KUKA KRL program: MyProgram_306().src

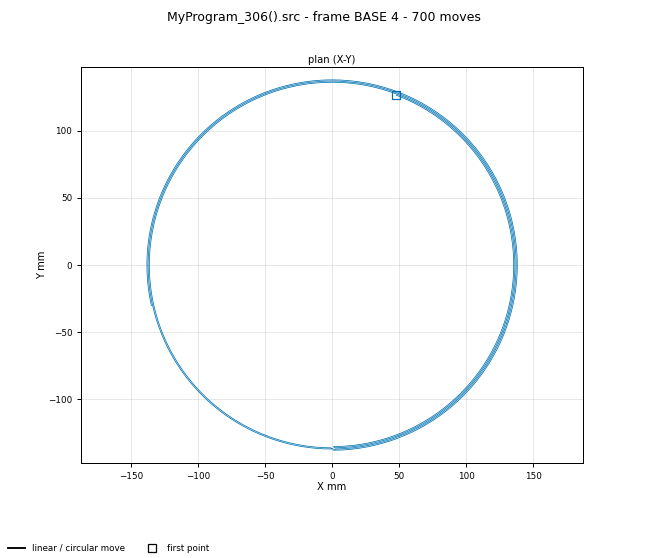
[picture p0: tool path of MyProgram_306().src in frame BASE 4, 700 of 700 moves have a stored position in this frame; points joined in program order, loops and branches not executed]
&ACCESS RVP
&REL 1
&PARAM TEMPLATE = C:\KRC\Roboter\Template\vorgabe
&PARAM EDITMASK = *
DEF MyProgram_306()
; ---- Setting reference (Base) ----
$BASE = BASE_DATA[4]

; --------------------------
; ---- Setting tool (TCP) ----
$TOOL = TOOL_DATA[3]
; --------------------------

$VEL.CP = VEL_APROX_PRINT
Startdeposition()
$VEL.CP = VEL_PRINT
LIN {X 47.8196,Y 126.5407,Z 181,A 70.0774,B 5.1523,C 0.0981,E1 5.2125,E2 382.635} C_DIS
LIN {X 50.7424,Y 125.3967,Z 181,A 68.7404,B 5.1523,C 0.0996,E1 5.216,E2 383.9727} C_DIS
LIN {X 53.7294,Y 124.1461,Z 181,A 67.3289,B 5.1523,C 0.1017,E1 5.2196,E2 385.3889} C_DIS
LIN {X 56.8494,Y 122.7487,Z 181,A 65.9585,B 5.1523,C 0.1025,E1 5.2231,E2 386.7498} C_DIS
LIN {X 60.1099,Y 121.1856,Z 181,A 64.4144,B 5.1522,C 0.1046,E1 5.227,E2 388.2953} C_DIS
LIN {X 63.2317,Y 119.5867,Z 181,A 62.9237,B 5.1522,C 0.1067,E1 5.2307,E2 389.7866} C_DIS
LIN {X 66.7997,Y 117.6329,Z 181,A 61.188,B 5.1522,C 0.1093,E1 5.2349,E2 391.5239} C_DIS
LIN {X 70.4878,Y 115.4608,Z 181,A 59.3984,B 5.152,C 0.1117,E1 5.2392,E2 393.3106} C_DIS
LIN {X 74.0978,Y 113.178,Z 181,A 57.6415,B 5.152,C 0.1139,E1 5.2433,E2 395.0613} C_DIS
LIN {X 77.4734,Y 110.8944,Z 181,A 55.903,B 5.152,C 0.1169,E1 5.2473,E2 396.8013} C_DIS
LIN {X 81.0975,Y 108.2727,Z 181,A 54.0011,B 5.1519,C 0.1202,E1 5.2516,E2 398.7043} C_DIS
LIN {X 84.4536,Y 105.6754,Z 181,A 52.2027,B 5.1518,C 0.1234,E1 5.2555,E2 400.5031} C_DIS
LIN {X 88.093,Y 102.6611,Z 181,A 50.2728,B 5.1518,C 0.1262,E1 5.2597,E2 402.4245} C_DIS
LIN {X 93.5773,Y 97.6879,Z 181,A 47.5115,B 5.1517,C 0.1274,E1 5.2653,E2 405.1411} C_DIS
LIN {X 95.6512,Y 95.6591,Z 181,A 45.6814,B 5.1514,C 0.1378,E1 5.269,E2 407.0442} C_DIS
LIN {X 98.4319,Y 92.7943,Z 181,A 44.4153,B 5.1514,C 0.1357,E1 5.2714,E2 408.2594} C_DIS
LIN {X 101.2138,Y 89.752,Z 181,A 42.6533,B 5.1514,C 0.1396,E1 5.2746,E2 410.0238} C_DIS
LIN {X 104.2851,Y 86.1641,Z 181,A 40.6959,B 5.1513,C 0.1434,E1 5.2782,E2 411.9765} C_DIS
LIN {X 107.3098,Y 82.3668,Z 181,A 38.7925,B 5.1512,C 0.146,E1 5.2814,E2 413.8619} C_DIS
LIN {X 109.5448,Y 79.3698,Z 181,A 37.1257,B 5.1511,C 0.1508,E1 5.2842,E2 415.5394} C_DIS
LIN {X 112.0158,Y 75.8426,Z 181,A 35.3544,B 5.151,C 0.1543,E1 5.287,E2 417.3049} C_DIS
LIN {X 114.5681,Y 71.9297,Z 181,A 33.411,B 5.1508,C 0.1586,E1 5.2899,E2 419.2447} C_DIS
LIN {X 116.9119,Y 68.0539,Z 181,A 31.5375,B 5.1507,C 0.1627,E1 5.2926,E2 421.1136} C_DIS
LIN {X 119.0066,Y 64.3209,Z 181,A 29.7725,B 5.1506,C 0.1666,E1 5.2949,E2 422.8735} C_DIS
LIN {X 120.8696,Y 60.7462,Z 181,A 28.2152,B 5.1505,C 0.1688,E1 5.2969,E2 424.4132} C_DIS
LIN {X 122.2077,Y 58.004,Z 181,A 26.919,B 5.1504,C 0.1722,E1 5.2985,E2 425.7104} C_DIS
LIN {X 123.801,Y 54.5253,Z 181,A 25.0947,B 5.1501,C 0.1792,E1 5.3006,E2 427.5605} C_DIS
LIN {X 126.0661,Y 49.0556,Z 181,A 22.9469,B 5.1501,C 0.1808,E1 5.3028,E2 429.6654} C_DIS
LIN {X 127.2877,Y 45.7925,Z 181,A 21.5116,B 5.15,C 0.1842,E1 5.3042,E2 431.0966} C_DIS
LIN {X 128.326,Y 42.7967,Z 181,A 20.1217,B 5.1498,C 0.1885,E1 5.3054,E2 432.493} C_DIS
LIN {X 129.3825,Y 39.4879,Z 181,A 18.7312,B 5.1498,C 0.1913,E1 5.3066,E2 433.8744} C_DIS
LIN {X 130.4088,Y 35.9572,Z 181,A 17.0921,B 5.1495,C 0.1967,E1 5.3078,E2 435.5245} C_DIS
LIN {X 131.5478,Y 31.5335,Z 181,A 15.4143,B 5.1495,C 0.1984,E1 5.3089,E2 437.1718} C_DIS
LIN {X 132.2174,Y 28.596,Z 181,A 14.092,B 5.1493,C 0.2026,E1 5.3098,E2 438.5006} C_DIS
LIN {X 132.966,Y 24.8892,Z 181,A 12.5495,B 5.1491,C 0.2063,E1 5.3106,E2 440.0369} C_DIS
LIN {X 133.6439,Y 20.9414,Z 181,A 10.8413,B 5.1489,C 0.2112,E1 5.3114,E2 441.7477} C_DIS
LIN {X 134.2991,Y 16.2171,Z 181,A 8.9489,B 5.1488,C 0.2151,E1 5.312,E2 443.6256} C_DIS
LIN {X 134.6572,Y 12.9089,Z 181,A 7.5424,B 5.1486,C 0.219,E1 5.3124,E2 445.0327} C_DIS
LIN {X 134.9389,Y 9.5299,Z 181,A 5.8041,B 5.1483,C 0.2274,E1 5.3128,E2 446.8094} C_DIS
LIN {X 135.1496,Y 5.844,Z 181,A 4.3625,B 5.1481,C 0.2301,E1 5.313,E2 448.2371} C_DIS
LIN {X 135.2694,Y 1.3606,Z 181,A 2.7211,B 5.1481,C 0.2318,E1 5.313,E2 449.8479} C_DIS
LIN {X 135.2556,Y -2.2721,Z 181,A 1.2724,B 5.1479,C 0.2349,E1 5.313,E2 451.2865} C_DIS
LIN {X 135.0337,Y -8.0739,Z 181,A -1.2689,B 5.1475,C 0.2431,E1 5.3127,E2 453.84} C_DIS
LIN {X 134.7703,Y -11.6735,Z 181,A -2.7066,B 5.1474,C 0.2461,E1 5.3124,E2 455.2676} C_DIS
LIN {X 134.3439,Y -15.8416,Z 181,A -4.3567,B 5.1472,C 0.2494,E1 5.3119,E2 456.9035} C_DIS
LIN {X 133.8283,Y -19.7368,Z 181,A -6.4275,B 5.1467,C 0.2599,E1 5.311,E2 459.0263} C_DIS
LIN {X 133.1281,Y -24.0026,Z 181,A -7.7215,B 5.1468,C 0.2574,E1 5.3104,E2 460.255} C_DIS
LIN {X 132.3167,Y -28.1358,Z 181,A -9.4984,B 5.1466,C 0.2623,E1 5.3094,E2 462.0325} C_DIS
LIN {X 131.4786,Y -31.8204,Z 181,A -11.0156,B 5.1464,C 0.2656,E1 5.3085,E2 463.5405} C_DIS
LIN {X 130.6362,Y -35.1196,Z 181,A -12.3908,B 5.1463,C 0.2686,E1 5.3075,E2 464.9085} C_DIS
LIN {X 129.7167,Y -38.3778,Z 181,A -13.8295,B 5.1461,C 0.2726,E1 5.3064,E2 466.349} C_DIS
LIN {X 128.511,Y -42.2412,Z 181,A -16.0648,B 5.1454,C 0.2847,E1 5.3044,E2 468.6509} C_DIS
LIN {X 126.8882,Y -46.8918,Z 181,A -17.9923,B 5.1452,C 0.2881,E1 5.3026,E2 470.5605} C_DIS
LIN {X 125.3399,Y -50.8835,Z 181,A -19.2432,B 5.1454,C 0.285,E1 5.3014,E2 471.7425} C_DIS
LIN {X 124.0945,Y -53.8487,Z 181,A -20.6394,B 5.1452,C 0.289,E1 5.2998,E2 473.1442} C_DIS
LIN {X 122.3624,Y -57.6803,Z 181,A -22.4382,B 5.1449,C 0.294,E1 5.2977,E2 474.9469} C_DIS
LIN {X 118.9552,Y -64.4163,Z 181,A -25.5886,B 5.1445,C 0.3015,E1 5.2937,E2 478.0942} C_DIS
LIN {X 116.6921,Y -68.4295,Z 181,A -27.4458,B 5.1442,C 0.3051,E1 5.2911,E2 479.9413} C_DIS
LIN {X 114.3467,Y -72.2804,Z 181,A -29.3004,B 5.144,C 0.309,E1 5.2884,E2 481.7906} C_DIS
LIN {X 111.8809,Y -76.0418,Z 181,A -31.1979,B 5.1437,C 0.3135,E1 5.2854,E2 483.6888} C_DIS
LIN {X 109.3024,Y -79.7042,Z 181,A -32.9951,B 5.1435,C 0.3166,E1 5.2825,E2 485.4751} C_DIS
LIN {X 106.7092,Y -83.1438,Z 181,A -34.8207,B 5.1433,C 0.3208,E1 5.2794,E2 487.3025} C_DIS
LIN {X 103.9092,Y -86.6181,Z 181,A -36.6922,B 5.143,C 0.3249,E1 5.2761,E2 489.1733} C_DIS
LIN {X 99.7215,Y -91.4073,Z 181,A -38.9686,B 5.143,C 0.325,E1 5.272,E2 491.399} C_DIS
LIN {X 97.7959,Y -93.4644,Z 181,A -40.4658,B 5.1426,C 0.3318,E1 5.2691,E2 492.9358} C_DIS
LIN {X 94.585,Y -96.7126,Z 181,A -42.9591,B 5.1418,C 0.3433,E1 5.264,E2 495.5013} C_DIS
LIN {X 90.6236,Y -100.4347,Z 181,A -44.5509,B 5.1422,C 0.3384,E1 5.2609,E2 497.0054} C_DIS
LIN {X 87.5053,Y -103.1623,Z 181,A -46.3354,B 5.1419,C 0.3422,E1 5.2571,E2 498.7951} C_DIS
LIN {X 83.9866,Y -106.0471,Z 181,A -48.2677,B 5.1417,C 0.3458,E1 5.2529,E2 500.7297} C_DIS
LIN {X 80.13,Y -108.99,Z 181,A -50.0733,B 5.1417,C 0.3462,E1 5.2489,E2 502.5053} C_DIS
LIN {X 77.226,Y -111.0666,Z 181,A -51.7178,B 5.1414,C 0.3506,E1 5.2451,E2 504.1679} C_DIS
LIN {X 73.5436,Y -113.5385,Z 181,A -53.5887,B 5.1411,C 0.3536,E1 5.2407,E2 506.0394} C_DIS
LIN {X 69.7824,Y -115.8883,Z 181,A -55.4441,B 5.141,C 0.3563,E1 5.2363,E2 507.8934} C_DIS
LIN {X 65.9154,Y -118.1311,Z 181,A -57.3271,B 5.1408,C 0.359,E1 5.2318,E2 509.7766} C_DIS
LIN {X 62.0394,Y -120.2113,Z 181,A -59.227,B 5.1406,C 0.3621,E1 5.227,E2 511.6825} C_DIS
LIN {X 58.8266,Y -121.8148,Z 181,A -60.449,B 5.1406,C 0.3603,E1 5.2241,E2 512.8676} C_DIS
LIN {X 56.384,Y -122.9639,Z 181,A -61.6646,B 5.1406,C 0.3628,E1 5.221,E2 514.0932} C_DIS
LIN {X 53.2137,Y -124.369,Z 181,A -63.6524,B 5.1399,C 0.3712,E1 5.2157,E2 516.148} C_DIS
LIN {X 49.0987,Y -126.0493,Z 181,A -65.111,B 5.1401,C 0.368,E1 5.212,E2 517.5542} C_DIS
LIN {X 44.5564,Y -127.7259,Z 181,A -67.1375,B 5.14,C 0.3699,E1 5.2067,E2 519.579} C_DIS
LIN {X 40.9196,Y -128.9371,Z 181,A -68.6696,B 5.14,C 0.3704,E1 5.2027,E2 521.1006} C_DIS
LIN {X 36.4436,Y -130.2728,Z 181,A -70.5721,B 5.14,C 0.3713,E1 5.1976,E2 522.9947} C_DIS
LIN {X 33.2477,Y -131.1249,Z 181,A -71.9881,B 5.1398,C 0.3726,E1 5.1938,E2 524.4135} C_DIS
LIN {X 29.9873,Y -131.9088,Z 181,A -73.3847,B 5.1398,C 0.3734,E1 5.19,E2 525.8079} C_DIS
LIN {X 26.8818,Y -132.5765,Z 181,A -74.6601,B 5.1398,C 0.3735,E1 5.1865,E2 527.0753} C_DIS
LIN {X 22.6495,Y -133.3654,Z 181,A -76.6157,B 5.1395,C 0.3763,E1 5.1811,E2 529.0489} C_DIS
LIN {X 18.9777,Y -133.9368,Z 181,A -78.1204,B 5.1395,C 0.3763,E1 5.1769,E2 530.5456} C_DIS
LIN {X 15.2137,Y -134.4184,Z 181,A -80.2974,B 5.139,C 0.3838,E1 5.1707,E2 532.796} C_DIS
LIN {X 10.4423,Y -134.8716,Z 181,A -81.8266,B 5.1394,C 0.3786,E1 5.1666,E2 534.2626} C_DIS
LIN {X 4.0171,Y -135.2153,Z 181,A -84.2235,B 5.1396,C 0.3755,E1 5.1601,E2 536.619} C_DIS
LIN {X 0.9559,Y -135.262,Z 181,A -86.2239,B 5.139,C 0.3838,E1 5.1542,E2 538.7094} C_DIS
Enddeposition()
LIN {X 0.9559,Y -135.262,Z 181,A -86.224,B 5.139,C 0.3838,E1 5.1542,E2 538.7095} C_DIS
Startdeposition()
$VEL.CP = VEL_PRINT
LIN {X 2.028,Y -136.1622,Z 181,A -83.6149,B 4.9954,C 0.3593,E1 5.017,E2 535.895} C_DIS
LIN {X 8.7445,Y -135.8964,Z 181,A -80.7975,B 4.9954,C 0.3585,E1 5.0248,E2 533.0777} C_DIS
LIN {X 15.4639,Y -135.2977,Z 181,A -78.8047,B 4.9948,C 0.3674,E1 5.0301,E2 531.1944} C_DIS
LIN {X 20.8523,Y -134.5708,Z 181,A -76.2066,B 4.9952,C 0.3624,E1 5.0374,E2 528.5544} C_DIS
LIN {X 24.8647,Y -133.8894,Z 181,A -74.8209,B 4.995,C 0.3653,E1 5.0411,E2 527.2105} C_DIS
LIN {X 28.4801,Y -133.1655,Z 181,A -73.3446,B 4.995,C 0.3651,E1 5.0451,E2 525.7429} C_DIS
LIN {X 31.9169,Y -132.3836,Z 181,A -71.9216,B 4.995,C 0.3647,E1 5.0489,E2 524.3268} C_DIS
LIN {X 34.7315,Y -131.6736,Z 181,A -70.6221,B 4.9951,C 0.3627,E1 5.0525,E2 523.0163} C_DIS
LIN {X 38.601,Y -130.5916,Z 181,A -68.9073,B 4.9953,C 0.3608,E1 5.0571,E2 521.2973} C_DIS
LIN {X 43.3333,Y -129.0984,Z 181,A -66.8158,B 4.9954,C 0.3587,E1 5.0626,E2 519.2039} C_DIS
LIN {X 46.4209,Y -128.0204,Z 181,A -64.8095,B 4.9961,C 0.3493,E1 5.0682,E2 517.114} C_DIS
LIN {X 51.9868,Y -125.8631,Z 181,A -62.9262,B 4.9957,C 0.3543,E1 5.0728,E2 515.3114} C_DIS
LIN {X 56.4258,Y -123.9387,Z 181,A -61.108,B 4.9957,C 0.3545,E1 5.0774,E2 513.5201} C_DIS
LIN {X 60.2896,Y -122.1032,Z 181,A -59.3056,B 4.9959,C 0.352,E1 5.0819,E2 511.716} C_DIS
LIN {X 63.7643,Y -120.3262,Z 181,A -57.6876,B 4.996,C 0.35,E1 5.0859,E2 510.0999} C_DIS
LIN {X 67.2784,Y -118.3987,Z 181,A -55.9698,B 4.9962,C 0.3471,E1 5.0901,E2 508.3767} C_DIS
LIN {X 70.8079,Y -116.3228,Z 181,A -54.2437,B 4.9964,C 0.3444,E1 5.0943,E2 506.6488} C_DIS
LIN {X 74.6135,Y -113.9189,Z 181,A -52.3601,B 4.9966,C 0.3414,E1 5.0987,E2 504.765} C_DIS
LIN {X 78.3293,Y -111.3963,Z 181,A -50.5287,B 4.9968,C 0.3389,E1 5.1029,E2 502.9397} C_DIS
LIN {X 82.4108,Y -108.4122,Z 181,A -48.4151,B 4.997,C 0.3353,E1 5.1076,E2 500.8262} C_DIS
LIN {X 85.9108,Y -105.66,Z 181,A -46.5831,B 4.9972,C 0.3324,E1 5.1116,E2 498.9979} C_DIS
LIN {X 89.293,Y -102.8175,Z 181,A -44.7681,B 4.9974,C 0.3294,E1 5.1154,E2 497.1871} C_DIS
LIN {X 92.3961,Y -100.0382,Z 181,A -42.6114,B 4.998,C 0.3204,E1 5.12,E2 494.9763} C_DIS
LIN {X 95.7918,Y -96.7914,Z 181,A -41.1149,B 4.9979,C 0.3229,E1 5.1228,E2 493.5406} C_DIS
LIN {X 98.8503,Y -93.6657,Z 181,A -39.085,B 4.9983,C 0.3164,E1 5.1268,E2 491.4845} C_DIS
LIN {X 101.2362,Y -91.0813,Z 181,A -37.8117,B 4.9983,C 0.316,E1 5.1291,E2 490.2368} C_DIS
LIN {X 104.3654,Y -87.4783,Z 181,A -35.9504,B 4.9985,C 0.3135,E1 5.1325,E2 488.3927} C_DIS
LIN {X 107.1144,Y -84.0897,Z 181,A -34.1474,B 4.9987,C 0.3098,E1 5.1356,E2 486.5924} C_DIS
LIN {X 109.7825,Y -80.5753,Z 181,A -32.3285,B 4.9989,C 0.306,E1 5.1387,E2 484.7766} C_DIS
LIN {X 112.2892,Y -77.0436,Z 181,A -30.5813,B 4.9991,C 0.3027,E1 5.1414,E2 483.0375} C_DIS
LIN {X 114.4748,Y -73.7581,Z 181,A -28.8977,B 4.9994,C 0.2983,E1 5.144,E2 481.3495} C_DIS
LIN {X 116.7973,Y -70.0222,Z 181,A -27.0852,B 4.9996,C 0.2943,E1 5.1467,E2 479.5403} C_DIS
LIN {X 119.0219,Y -66.1697,Z 181,A -25.3167,B 4.9998,C 0.291,E1 5.1491,E2 477.7835} C_DIS
LIN {X 121.408,Y -61.6777,Z 181,A -23.1686,B 5.0001,C 0.2854,E1 5.1518,E2 475.6324} C_DIS
LIN {X 123.5611,Y -57.2423,Z 181,A -21.2809,B 5.0003,C 0.2826,E1 5.1541,E2 473.7669} C_DIS
LIN {X 124.947,Y -54.1506,Z 181,A -19.8732,B 5.0005,C 0.2791,E1 5.1557,E2 472.3603} C_DIS
LIN {X 126.753,Y -49.7791,Z 181,A -17.954,B 5.0007,C 0.2748,E1 5.1577,E2 470.4485} C_DIS
LIN {X 127.8654,Y -46.8507,Z 181,A -16.3001,B 5.0012,C 0.2665,E1 5.1593,E2 468.7504} C_DIS
LIN {X 129.0515,Y -43.4741,Z 181,A -15.1153,B 5.0012,C 0.267,E1 5.1603,E2 467.6055} C_DIS
LIN {X 129.983,Y -40.6093,Z 181,A -13.8576,B 5.0013,C 0.2637,E1 5.1614,E2 466.3481} C_DIS
LIN {X 131.1503,Y -36.6564,Z 181,A -12.319,B 5.0014,C 0.2617,E1 5.1626,E2 464.833} C_DIS
LIN {X 131.9747,Y -33.5676,Z 181,A -10.9179,B 5.0017,C 0.2572,E1 5.1636,E2 463.4236} C_DIS
LIN {X 132.9297,Y -29.57,Z 181,A -9.1267,B 5.002,C 0.2515,E1 5.1647,E2 461.6232} C_DIS
LIN {X 133.7363,Y -25.6657,Z 181,A -7.6166,B 5.002,C 0.2491,E1 5.1655,E2 460.1329} C_DIS
LIN {X 134.2964,Y -22.5524,Z 181,A -5.9168,B 5.0025,C 0.2401,E1 5.1663,E2 458.3849} C_DIS
LIN {X 134.9324,Y -18.3813,Z 181,A -4.5365,B 5.0025,C 0.2408,E1 5.1668,E2 457.0538} C_DIS
LIN {X 135.3989,Y -14.5361,Z 181,A -3.0388,B 5.0026,C 0.238,E1 5.1673,E2 455.5716} C_DIS
LIN {X 135.8912,Y -8.83,Z 181,A 0.0247,B 5.0034,C 0.2218,E1 5.1679,E2 452.4226} C_DIS
LIN {X 136.1441,Y -3.0766,Z 181,A 1.6633,B 5.0032,C 0.2262,E1 5.1681,E2 450.8826} C_DIS
LIN {X 136.1281,Y 3.6531,Z 181,A 4.3463,B 5.0034,C 0.2202,E1 5.168,E2 448.2163} C_DIS
LIN {X 135.7749,Y 10.4711,Z 181,A 7.2923,B 5.0038,C 0.211,E1 5.1675,E2 445.2591} C_DIS
LIN {X 135.4246,Y 14.2965,Z 181,A 8.8988,B 5.004,C 0.2066,E1 5.1671,E2 443.6527} C_DIS
LIN {X 134.8881,Y 18.6989,Z 181,A 10.6539,B 5.0042,C 0.2029,E1 5.1664,E2 441.9104} C_DIS
LIN {X 134.3507,Y 22.2269,Z 181,A 12.0546,B 5.0042,C 0.2001,E1 5.1658,E2 440.5215} C_DIS
LIN {X 133.7488,Y 25.6004,Z 181,A 13.4568,B 5.0044,C 0.1966,E1 5.1651,E2 439.1232} C_DIS
LIN {X 133.0564,Y 28.9857,Z 181,A 14.8859,B 5.0045,C 0.1929,E1 5.1643,E2 437.6964} C_DIS
LIN {X 132.1674,Y 32.808,Z 181,A 16.5738,B 5.0047,C 0.1879,E1 5.1632,E2 436.0029} C_DIS
LIN {X 131.1408,Y 36.6902,Z 181,A 18.1184,B 5.0048,C 0.1853,E1 5.162,E2 434.4755} C_DIS
LIN {X 130.1423,Y 40.0888,Z 181,A 19.4608,B 5.0049,C 0.1833,E1 5.161,E2 433.1507} C_DIS
LIN {X 129.2623,Y 42.8413,Z 181,A 20.7675,B 5.0051,C 0.1787,E1 5.1598,E2 431.832} C_DIS
LIN {X 128.2866,Y 45.6824,Z 181,A 22.035,B 5.0051,C 0.1753,E1 5.1587,E2 430.5634} C_DIS
LIN {X 127.2782,Y 48.4233,Z 181,A 23.2607,B 5.0053,C 0.1721,E1 5.1575,E2 429.3375} C_DIS
LIN {X 124.7033,Y 54.7143,Z 181,A 26.0669,B 5.0055,C 0.1653,E1 5.1544,E2 426.5366} C_DIS
LIN {X 123.0236,Y 58.3895,Z 181,A 27.6576,B 5.0056,C 0.1624,E1 5.1526,E2 424.9588} C_DIS
LIN {X 121.5759,Y 61.3479,Z 181,A 29.0819,B 5.0058,C 0.1584,E1 5.1508,E2 423.529} C_DIS
LIN {X 119.7296,Y 64.881,Z 181,A 30.7364,B 5.0058,C 0.1545,E1 5.1486,E2 421.8768} C_DIS
LIN {X 117.484,Y 68.8629,Z 181,A 32.5741,B 5.006,C 0.1509,E1 5.1461,E2 420.049} C_DIS
LIN {X 115.1475,Y 72.7023,Z 181,A 34.4188,B 5.0061,C 0.147,E1 5.1434,E2 418.2094} C_DIS
LIN {X 112.6971,Y 76.4458,Z 181,A 36.2084,B 5.0061,C 0.1438,E1 5.1406,E2 416.4306} C_DIS
LIN {X 110.2737,Y 79.9017,Z 181,A 37.9643,B 5.0063,C 0.1399,E1 5.1378,E2 414.6765} C_DIS
LIN {X 107.9936,Y 82.9581,Z 181,A 39.555,B 5.0064,C 0.1364,E1 5.1351,E2 413.0871} C_DIS
LIN {X 105.1893,Y 86.486,Z 181,A 41.4629,B 5.0065,C 0.1321,E1 5.1317,E2 411.1772} C_DIS
LIN {X 102.1937,Y 90.0061,Z 181,A 43.3409,B 5.0066,C 0.1287,E1 5.1283,E2 409.3069} C_DIS
LIN {X 99.5883,Y 92.8803,Z 181,A 45.3778,B 5.0068,C 0.12,E1 5.1243,E2 407.2193} C_DIS
LIN {X 96.2668,Y 96.3195,Z 181,A 46.6425,B 5.0067,C 0.1257,E1 5.122,E2 406.047} C_DIS
LIN {X 91.2692,Y 101.0674,Z 181,A 49.7341,B 5.0069,C 0.1175,E1 5.1157,E2 402.9314} C_DIS
LIN {X 87.9494,Y 103.9692,Z 181,A 51.443,B 5.0069,C 0.1159,E1 5.1121,E2 401.2403} C_DIS
LIN {X 84.7506,Y 106.5923,Z 181,A 53.3248,B 5.007,C 0.111,E1 5.108,E2 399.3409} C_DIS
LIN {X 80.9544,Y 109.504,Z 181,A 55.2605,B 5.007,C 0.1085,E1 5.1037,E2 397.4146} C_DIS
LIN {X 77.3453,Y 112.0821,Z 181,A 57.1065,B 5.0071,C 0.1056,E1 5.0994,E2 395.571} C_DIS
LIN {X 73.474,Y 114.6567,Z 181,A 58.9776,B 5.0071,C 0.1036,E1 5.0951,E2 393.7102} C_DIS
LIN {X 69.8678,Y 116.8893,Z 181,A 60.7644,B 5.0072,C 0.1009,E1 5.0908,E2 391.9232} C_DIS
LIN {X 65.9745,Y 119.13,Z 181,A 62.611,B 5.0072,C 0.0987,E1 5.0863,E2 390.082} C_DIS
LIN {X 62.1791,Y 121.1527,Z 181,A 64.2799,B 5.0073,C 0.0979,E1 5.0823,E2 388.4304} C_DIS
LIN {X 58.9076,Y 122.7761,Z 181,A 65.851,B 5.0073,C 0.0956,E1 5.0783,E2 386.8552} C_DIS
LIN {X 56.0284,Y 124.1172,Z 181,A 67.1928,B 5.0073,C 0.0939,E1 5.0749,E2 385.5128} C_DIS
LIN {X 52.6663,Y 125.58,Z 181,A 68.5818,B 5.0073,C 0.0939,E1 5.0714,E2 384.1429} C_DIS
LIN {X 49.5594,Y 126.8384,Z 181,A 70.0541,B 5.0074,C 0.0916,E1 5.0675,E2 382.6631} C_DIS
LIN {X 47.0293,Y 127.8003,Z 181,A 71.3451,B 5.0074,C 0.0887,E1 5.0641,E2 381.3537} C_DIS
LIN {X 43.2842,Y 129.1148,Z 181,A 72.8823,B 5.0074,C 0.0887,E1 5.0601,E2 379.8331} C_DIS
LIN {X 36.771,Y 131.1182,Z 181,A 75.6055,B 5.0074,C 0.0878,E1 5.0529,E2 377.1281} C_DIS
LIN {X 33.6246,Y 131.9602,Z 181,A 77.051,B 5.0075,C 0.0859,E1 5.0489,E2 375.6738} C_DIS
LIN {X 30.1633,Y 132.7942,Z 181,A 78.5411,B 5.0075,C 0.085,E1 5.0449,E2 374.1851} C_DIS
LIN {X 26.4413,Y 133.587,Z 181,A 80.2021,B 5.0075,C 0.0833,E1 5.0403,E2 372.5172} C_DIS
LIN {X 22.8669,Y 134.244,Z 181,A 81.6663,B 5.0075,C 0.0833,E1 5.0363,E2 371.0615} C_DIS
LIN {X 19.5681,Y 134.7639,Z 181,A 83.0717,B 5.0075,C 0.0825,E1 5.0324,E2 369.6564} C_DIS
LIN {X 14.042,Y 135.452,Z 181,A 85.8196,B 5.0077,C 0.0772,E1 5.0247,E2 366.8599} C_DIS
LIN {X 10.059,Y 135.805,Z 181,A 87.0891,B 5.0077,C 0.0813,E1 5.0213,E2 365.6414} C_DIS
LIN {X 6.0667,Y 136.0439,Z 181,A 88.9885,B 5.0077,C 0.0786,E1 5.0159,E2 363.7163} C_DIS
LIN {X 1.3417,Y 136.1717,Z 181,A 91.4927,B 5.0077,C 0.0728,E1 5.0087,E2 361.1496} C_DIS
LIN {X -4.4974,Y 136.1046,Z 181,A 93.2988,B 5.0077,C 0.0799,E1 5.0039,E2 359.4247} C_DIS
LIN {X -10.7726,Y 135.7519,Z 181,A 96.3123,B 5.0077,C 0.0764,E1 4.9954,E2 356.3672} C_DIS
LIN {X -14.954,Y 135.3539,Z 181,A 97.6002,B 5.0076,C 0.0818,E1 4.992,E2 355.1389} C_DIS
LIN {X -18.7034,Y 134.8875,Z 181,A 99.2311,B 5.0076,C 0.0818,E1 4.9874,E2 353.5038} C_DIS
LIN {X -22.171,Y 134.3601,Z 181,A 100.6494,B 5.0076,C 0.0831,E1 4.9835,E2 352.0934} C_DIS
LIN {X -25.0922,Y 133.8459,Z 181,A 102.0094,B 5.0076,C 0.0825,E1 4.9798,E2 350.7204} C_DIS
LIN {X -28.7373,Y 133.11,Z 181,A 103.5032,B 5.0076,C 0.084,E1 4.9757,E2 349.2361} C_DIS
LIN {X -32.2356,Y 132.3067,Z 181,A 105.1023,B 5.0076,C 0.084,E1 4.9713,E2 347.6271} C_DIS
LIN {X -36.4872,Y 131.1976,Z 181,A 106.6379,B 5.0075,C 0.0884,E1 4.9673,E2 346.1307} C_DIS
LIN {X -39.6732,Y 130.2695,Z 181,A 108.3833,B 5.0075,C 0.0861,E1 4.9625,E2 344.3437} C_DIS
LIN {X -43.2649,Y 129.1212,Z 181,A 110.591,B 5.0075,C 0.0814,E1 4.9565,E2 342.0609} C_DIS
LIN {X -48.3963,Y 127.288,Z 181,A 112.3107,B 5.0075,C 0.0891,E1 4.9522,E2 340.4131} C_DIS
LIN {X -52.1404,Y 125.7997,Z 181,A 114.1747,B 5.0075,C 0.0892,E1 4.9473,E2 338.5296} C_DIS
LIN {X -56.8583,Y 123.7387,Z 181,A 116.1105,B 5.0074,C 0.0939,E1 4.9424,E2 336.6234} C_DIS
LIN {X -59.8078,Y 122.3409,Z 181,A 117.364,B 5.0074,C 0.0966,E1 4.9393,E2 335.3855} C_DIS
LIN {X -63.4973,Y 120.4664,Z 181,A 119.2161,B 5.0074,C 0.0978,E1 4.9347,E2 333.5212} C_DIS
LIN {X -67.1669,Y 118.4623,Z 181,A 121.1697,B 5.0073,C 0.0984,E1 4.9299,E2 331.5453} C_DIS
LIN {X -70.156,Y 116.717,Z 181,A 123.3369,B 5.0073,C 0.094,E1 4.9245,E2 329.2918} C_DIS
LIN {X -75.1856,Y 113.5422,Z 181,A 125.1812,B 5.0072,C 0.1038,E1 4.9204,E2 327.5305} C_DIS
LIN {X -78.9167,Y 110.9813,Z 181,A 127.1414,B 5.0072,C 0.1063,E1 4.9159,E2 325.5648} C_DIS
LIN {X -82.5442,Y 108.3101,Z 181,A 129.0557,B 5.0071,C 0.1093,E1 4.9116,E2 323.6497} C_DIS
LIN {X -86.2039,Y 105.4204,Z 181,A 131.018,B 5.007,C 0.1127,E1 4.9073,E2 321.689} C_DIS
LIN {X -89.7058,Y 102.4573,Z 181,A 132.9817,B 5.007,C 0.116,E1 4.9031,E2 319.7227} C_DIS
LIN {X -93.0511,Y 99.4293,Z 181,A 134.922,B 5.0068,C 0.1192,E1 4.8991,E2 317.7789} C_DIS
LIN {X -96.1912,Y 96.3945,Z 181,A 136.8167,B 5.0068,C 0.1224,E1 4.8954,E2 315.8786} C_DIS
LIN {X -99.3695,Y 93.1153,Z 181,A 138.8079,B 5.0067,C 0.1257,E1 4.8915,E2 313.8805} C_DIS
LIN {X -102.4157,Y 89.7534,Z 181,A 140.7423,B 5.0066,C 0.1295,E1 4.8879,E2 311.9445} C_DIS
LIN {X -105.3382,Y 86.3045,Z 181,A 142.6805,B 5.0065,C 0.1333,E1 4.8844,E2 310.0035} C_DIS
LIN {X -108.1861,Y 82.7063,Z 181,A 144.6358,B 5.0064,C 0.1374,E1 4.8811,E2 308.0467} C_DIS
LIN {X -110.9394,Y 78.9753,Z 181,A 146.5997,B 5.0063,C 0.1418,E1 4.8779,E2 306.083} C_DIS
LIN {X -113.6721,Y 74.9883,Z 181,A 149.153,B 5.0063,C 0.1423,E1 4.8738,E2 303.4671} C_DIS
LIN {X -116.0563,Y 71.2427,Z 181,A 151.3666,B 5.0062,C 0.144,E1 4.8705,E2 301.2121} C_DIS
LIN {X -119.0798,Y 66.0651,Z 181,A 152.8445,B 5.0057,C 0.1587,E1 4.8687,E2 299.8659} C_DIS
LIN {X -122.4558,Y 59.5748,Z 181,A 156.4438,B 5.0057,C 0.1624,E1 4.864,E2 296.2053} C_DIS
LIN {X -124.2151,Y 55.8094,Z 181,A 158.0634,B 5.0054,C 0.1679,E1 4.8621,E2 294.603} C_DIS
LIN {X -125.5427,Y 52.7558,Z 181,A 159.5086,B 5.0054,C 0.1712,E1 4.8606,E2 293.1535} C_DIS
LIN {X -126.8119,Y 49.6274,Z 181,A 160.9595,B 5.0052,C 0.1747,E1 4.8591,E2 291.7001} C_DIS
LIN {X -127.8506,Y 46.8918,Z 181,A 162.6374,B 5.0052,C 0.1745,E1 4.8574,E2 289.9679} C_DIS
LIN {X -129.0498,Y 43.4794,Z 181,A 164.0283,B 5.005,C 0.1796,E1 4.8562,E2 288.5944} C_DIS
LIN {X -130.4176,Y 39.1894,Z 181,A 165.7654,B 5.0048,C 0.186,E1 4.8547,E2 286.8786} C_DIS
LIN {X -131.7967,Y 34.2687,Z 181,A 168.1146,B 5.0046,C 0.1904,E1 4.853,E2 284.5064} C_DIS
LIN {X -132.6329,Y 30.8694,Z 181,A 169.5985,B 5.0045,C 0.1944,E1 4.8521,E2 283.0223} C_DIS
LIN {X -133.3798,Y 27.4599,Z 181,A 171.0105,B 5.0043,C 0.1989,E1 4.8512,E2 281.6186} C_DIS
LIN {X -133.9577,Y 24.4892,Z 181,A 172.3852,B 5.0043,C 0.2017,E1 4.8505,E2 280.2323} C_DIS
LIN {X -134.5709,Y 20.8516,Z 181,A 173.8946,B 5.004,C 0.2063,E1 4.8499,E2 278.7294} C_DIS
LIN {X -135.0492,Y 17.4897,Z 181,A 175.4363,B 5.0039,C 0.2095,E1 4.8493,E2 277.1748} C_DIS
LIN {X -135.5373,Y 13.1839,Z 181,A 177.2749,B 5.0037,C 0.2145,E1 4.8487,E2 275.3357} C_DIS
LIN {X -135.8459,Y 9.4985,Z 181,A 178.9934,B 5.0035,C 0.2177,E1 4.8484,E2 273.5981} C_DIS
LIN {X -136.0728,Y 5.3259,Z 181,A -179.3077,B 5.0033,C 0.2231,E1 4.8482,E2 271.9079} C_DIS
LIN {X -136.17,Y 1.5593,Z 181,A -177.5443,B 5.0032,C 0.2263,E1 4.8481,E2 270.1235} C_DIS
LIN {X -136.1533,Y -2.5594,Z 181,A -175.861,B 5.0029,C 0.2316,E1 4.8481,E2 268.4476} C_DIS
LIN {X -136.0155,Y -6.6325,Z 181,A -174.1816,B 5.0027,C 0.2367,E1 4.8483,E2 266.7738} C_DIS
LIN {X -135.815,Y -9.9228,Z 181,A -172.7078,B 5.0025,C 0.24,E1 4.8486,E2 265.2902} C_DIS
LIN {X -135.4612,Y -13.9571,Z 181,A -170.8732,B 5.0023,C 0.2437,E1 4.8491,E2 263.4403} C_DIS
LIN {X -135.0123,Y -17.7712,Z 181,A -169.2336,B 5.0021,C 0.2481,E1 4.8497,E2 261.7988} C_DIS
LIN {X -134.3689,Y -22.1182,Z 181,A -167.3782,B 5.0019,C 0.2532,E1 4.8504,E2 259.9438} C_DIS
LIN {X -133.772,Y -25.4791,Z 181,A -165.937,B 5.0017,C 0.2572,E1 4.8512,E2 258.5029} C_DIS
LIN {X -133.1026,Y -28.7716,Z 181,A -164.4669,B 5.0015,C 0.2607,E1 4.852,E2 257.0266} C_DIS
LIN {X -132.4755,Y -31.5356,Z 181,A -162.5842,B 5.0016,C 0.2584,E1 4.8533,E2 255.0571} C_DIS
LIN {X -131.2171,Y -36.4175,Z 181,A -160.9064,B 5.0011,C 0.2678,E1 4.8545,E2 253.437} C_DIS
LIN {X -129.6663,Y -41.6024,Z 181,A -158.7242,B 5.0007,C 0.2747,E1 4.8563,E2 251.2681} C_DIS
LIN {X -128.6253,Y -44.7171,Z 181,A -156.8852,B 5.0007,C 0.2747,E1 4.858,E2 249.3717} C_DIS
LIN {X -127.2958,Y -48.3763,Z 181,A -155.4454,B 5.0004,C 0.2806,E1 4.8594,E2 247.9582} C_DIS
LIN {X -125.7785,Y -52.191,Z 181,A -153.8187,B 5.0001,C 0.2859,E1 4.8611,E2 246.3451} C_DIS
LIN {X -124.4431,Y -55.2998,Z 181,A -152.3226,B 4.9999,C 0.289,E1 4.8628,E2 244.8405} C_DIS
LIN {X -122.8053,Y -58.8466,Z 181,A -150.6586,B 4.9997,C 0.293,E1 4.8648,E2 243.1747} C_DIS
LIN {X -121.2541,Y -61.9799,Z 181,A -149.1568,B 4.9995,C 0.2964,E1 4.8667,E2 241.6696} C_DIS
LIN {X -119.7911,Y -64.7674,Z 181,A -147.2356,B 4.9996,C 0.2946,E1 4.8693,E2 239.6728} C_DIS
LIN {X -117.4959,Y -68.8427,Z 181,A -145.6876,B 4.9991,C 0.3029,E1 4.8714,E2 238.1795} C_DIS
LIN {X -115.0896,Y -72.7941,Z 181,A -143.7565,B 4.9988,C 0.3077,E1 4.8742,E2 236.2512} C_DIS
LIN {X -112.842,Y -76.2317,Z 181,A -141.9154,B 4.9986,C 0.3107,E1 4.8771,E2 234.3962} C_DIS
LIN {X -110.1528,Y -80.0686,Z 181,A -139.939,B 4.9984,C 0.3151,E1 4.8803,E2 232.4198} C_DIS
LIN {X -107.472,Y -83.6326,Z 181,A -138.0383,B 4.9981,C 0.319,E1 4.8835,E2 230.5166} C_DIS
LIN {X -104.8947,Y -86.8428,Z 181,A -136.2259,B 4.9979,C 0.322,E1 4.8868,E2 228.6944} C_DIS
LIN {X -101.9076,Y -90.3297,Z 181,A -134.3245,B 4.9976,C 0.3263,E1 4.8902,E2 226.7974} C_DIS
LIN {X -98.6538,Y -93.8728,Z 181,A -132.1493,B 4.9975,C 0.329,E1 4.8944,E2 224.6033} C_DIS
LIN {X -95.9508,Y -96.6334,Z 181,A -130.5,B 4.9973,C 0.332,E1 4.8977,E2 222.9512} C_DIS
LIN {X -92.6368,Y -99.8151,Z 181,A -128.5648,B 4.997,C 0.3356,E1 4.9016,E2 221.0161} C_DIS
LIN {X -89.3479,Y -102.7696,Z 181,A -126.6278,B 4.9969,C 0.3382,E1 4.9057,E2 219.0695} C_DIS
LIN {X -85.7901,Y -105.7581,Z 181,A -124.6683,B 4.9966,C 0.3415,E1 4.9099,E2 217.1096} C_DIS
LIN {X -82.4497,Y -108.3824,Z 181,A -122.8444,B 4.9965,C 0.3441,E1 4.914,E2 215.2812} C_DIS
LIN {X -78.9142,Y -110.9831,Z 181,A -120.9454,B 4.9963,C 0.3465,E1 4.9183,E2 213.3755} C_DIS
LIN {X -75.1587,Y -113.5599,Z 181,A -119.0292,B 4.9961,C 0.3494,E1 4.9227,E2 211.4594} C_DIS
LIN {X -71.7177,Y -115.7636,Z 181,A -117.2752,B 4.9959,C 0.3515,E1 4.9269,E2 209.7009} C_DIS
LIN {X -67.9022,Y -118.0424,Z 181,A -115.3784,B 4.9958,C 0.3537,E1 4.9315,E2 207.8006} C_DIS
LIN {X -64.07,Y -120.1657,Z 181,A -113.4315,B 4.9957,C 0.355,E1 4.9363,E2 205.8401} C_DIS
LIN {X -60.3358,Y -122.0804,Z 181,A -111.8521,B 4.9954,C 0.3589,E1 4.9401,E2 204.2846} C_DIS
LIN {X -57.5962,Y -123.3975,Z 181,A -110.4697,B 4.9954,C 0.3593,E1 4.9437,E2 202.8887} C_DIS
LIN {X -54.358,Y -124.8574,Z 181,A -109.017,B 4.9952,C 0.3612,E1 4.9474,E2 201.4413} C_DIS
LIN {X -51.1421,Y -126.2085,Z 181,A -107.7619,B 4.995,C 0.3648,E1 4.9505,E2 200.2135} C_DIS
LIN {X -47.907,Y -127.4715,Z 181,A -106.0884,B 4.995,C 0.364,E1 4.955,E2 198.5123} C_DIS
LIN {X -43.72,Y -128.9696,Z 181,A -103.6748,B 4.9953,C 0.3599,E1 4.9615,E2 196.0278} C_DIS
LIN {X -39.6364,Y -130.2808,Z 181,A -102.3646,B 4.9949,C 0.3663,E1 4.9649,E2 194.7816} C_DIS
LIN {X -35.815,Y -131.3847,Z 181,A -100.5454,B 4.9949,C 0.3659,E1 4.9698,E2 192.9431} C_DIS
LIN {X -32.4742,Y -132.2492,Z 181,A -99.1496,B 4.9949,C 0.3673,E1 4.9736,E2 191.5542} C_DIS
LIN {X -28.9633,Y -133.0612,Z 181,A -97.7191,B 4.9947,C 0.369,E1 4.9774,E2 190.1343} C_DIS
LIN {X -25.9914,Y -133.674,Z 181,A -96.3647,B 4.9947,C 0.3687,E1 4.9812,E2 188.7694} C_DIS
LIN {X -22.429,Y -134.317,Z 181,A -94.9142,B 4.9947,C 0.37,E1 4.9852,E2 187.3278} C_DIS
LIN {X -19.3327,Y -134.7976,Z 181,A -93.2365,B 4.9949,C 0.3664,E1 4.9899,E2 185.6028} C_DIS
LIN {X -15.9037,Y -135.2452,Z 181,A -91.7796,B 4.9949,C 0.3667,E1 4.994,E2 184.1451} C_DIS
LIN {X -12.3874,Y -135.6138,Z 181,A -90.6397,B 4.9945,C 0.3708,E1 4.997,E2 183.0501} C_DIS
LIN {X -6.9591,Y -135.9991,Z 181,A -88.3319,B 4.9945,C 0.3708,E1 5.0035,E2 180.739} C_DIS
LIN {X -1.0575,Y -136.1733,Z 181,A -85.7858,B 4.9946,C 0.3699,E1 5.0106,E2 178.1837} C_DIS
LIN {X -1.0575,Y -136.1733,Z 181,A -85.7858,B 4.9946,C 0.3699,E1 5.0106,E2 178.1837} C_DIS
Enddeposition()
LIN {X 0.9703,Y -137.0729,Z 181,A -85.3499,B 4.954,C 0.3766,E1 4.9715,E2 177.845} C_DIS
Startdeposition()
$VEL.CP = VEL_PRINT
LIN {X -3.0365,Y -137.0479,Z 181,A -87.2094,B 4.9538,C 0.3788,E1 4.9662,E2 179.7296} C_DIS
LIN {X -5.9106,Y -136.9531,Z 181,A -88.6175,B 4.9536,C 0.3811,E1 4.9622,E2 181.1649} C_DIS
LIN {X -12.2339,Y -136.5341,Z 181,A -91.0466,B 4.9538,C 0.3785,E1 4.9555,E2 183.5666} C_DIS
LIN {X -17.3238,Y -135.981,Z 181,A -93.2409,B 4.9538,C 0.3787,E1 4.9494,E2 185.7688} C_DIS
LIN {X -23.0386,Y -135.1302,Z 181,A -95.6152,B 4.9539,C 0.3775,E1 4.9429,E2 188.1387} C_DIS
LIN {X -26.0662,Y -134.5784,Z 181,A -97.0589,B 4.9539,C 0.3787,E1 4.9389,E2 189.6032} C_DIS
LIN {X -29.9261,Y -133.774,Z 181,A -98.5216,B 4.954,C 0.3759,E1 4.9349,E2 191.0425} C_DIS
LIN {X -32.4324,Y -133.1875,Z 181,A -99.6375,B 4.954,C 0.3758,E1 4.9319,E2 192.1638} C_DIS
LIN {X -35.4722,Y -132.41,Z 181,A -101.0196,B 4.954,C 0.3758,E1 4.9281,E2 193.5553} C_DIS
LIN {X -39.1587,Y -131.3685,Z 181,A -102.7675,B 4.954,C 0.3762,E1 4.9234,E2 195.3227} C_DIS
LIN {X -43.4499,Y -130.0107,Z 181,A -104.5928,B 4.9542,C 0.3742,E1 4.9185,E2 197.141} C_DIS
LIN {X -46.9529,Y -128.7878,Z 181,A -106.0851,B 4.9543,C 0.3723,E1 4.9146,E2 198.6262} C_DIS
LIN {X -50.7356,Y -127.3453,Z 181,A -107.6804,B 4.9545,C 0.3698,E1 4.9105,E2 200.2092} C_DIS
LIN {X -53.3815,Y -126.2592,Z 181,A -108.9727,B 4.9545,C 0.3696,E1 4.9072,E2 201.5142} C_DIS
LIN {X -56.1546,Y -125.0492,Z 181,A -110.2932,B 4.9545,C 0.3688,E1 4.9038,E2 202.842} C_DIS
LIN {X -59.3857,Y -123.5478,Z 181,A -111.8122,B 4.9547,C 0.3675,E1 4.8999,E2 204.3651} C_DIS
LIN {X -63.2167,Y -121.633,Z 181,A -113.6539,B 4.9547,C 0.3659,E1 4.8953,E2 206.2135} C_DIS
LIN {X -67.0731,Y -119.5507,Z 181,A -115.5503,B 4.9549,C 0.3642,E1 4.8906,E2 208.1184} C_DIS
LIN {X -71.1164,Y -117.1907,Z 181,A -117.54,B 4.9551,C 0.3619,E1 4.8859,E2 210.1124} C_DIS
LIN {X -74.9995,Y -114.745,Z 181,A -119.5177,B 4.9552,C 0.3597,E1 4.8812,E2 212.0977} C_DIS
LIN {X -78.7321,Y -112.2165,Z 181,A -121.3976,B 4.9554,C 0.3568,E1 4.8769,E2 213.977} C_DIS
LIN {X -82.2272,Y -109.6815,Z 181,A -123.2429,B 4.9556,C 0.3543,E1 4.8727,E2 215.8273} C_DIS
LIN {X -85.7952,Y -106.9133,Z 181,A -125.1986,B 4.9558,C 0.3518,E1 4.8684,E2 217.7916} C_DIS
LIN {X -90.1845,Y -103.2372,Z 181,A -127.3722,B 4.9562,C 0.3456,E1 4.8638,E2 219.9367} C_DIS
LIN {X -92.7464,Y -100.9418,Z 181,A -129.0711,B 4.9562,C 0.3453,E1 4.8602,E2 221.6689} C_DIS
LIN {X -96.068,Y -97.786,Z 181,A -131.0795,B 4.9564,C 0.3425,E1 4.8562,E2 223.6889} C_DIS
LIN {X -99.2626,Y -94.5417,Z 181,A -133.5232,B 4.9564,C 0.3435,E1 4.8514,E2 226.2009} C_DIS
LIN {X -102.8064,Y -90.6754,Z 181,A -135.1709,B 4.957,C 0.3343,E1 4.8484,E2 227.7789} C_DIS
LIN {X -105.7793,Y -87.1894,Z 181,A -137.1285,B 4.9573,C 0.3306,E1 4.8449,E2 229.7414} C_DIS
LIN {X -108.5828,Y -83.6725,Z 181,A -139.0869,B 4.9575,C 0.3272,E1 4.8415,E2 231.7093} C_DIS
LIN {X -111.1938,Y -80.1699,Z 181,A -140.8842,B 4.9578,C 0.3228,E1 4.8385,E2 233.5024} C_DIS
LIN {X -113.6671,Y -76.6226,Z 181,A -142.7192,B 4.958,C 0.3189,E1 4.8356,E2 235.3402} C_DIS
LIN {X -115.9919,Y -73.0551,Z 181,A -144.5963,B 4.9582,C 0.3156,E1 4.8328,E2 237.229} C_DIS
LIN {X -118.3582,Y -69.1564,Z 181,A -146.66,B 4.9584,C 0.3123,E1 4.8298,E2 239.3119} C_DIS
LIN {X -120.702,Y -64.9784,Z 181,A -148.7085,B 4.9587,C 0.3078,E1 4.827,E2 241.3654} C_DIS
LIN {X -122.5672,Y -61.3887,Z 181,A -150.4464,B 4.959,C 0.304,E1 4.8248,E2 243.1085} C_DIS
LIN {X -124.5369,Y -57.2822,Z 181,A -152.2228,B 4.9593,C 0.2981,E1 4.8227,E2 244.8678} C_DIS
LIN {X -125.9793,Y -54.0369,Z 181,A -153.7819,B 4.9595,C 0.2949,E1 4.821,E2 246.4357} C_DIS
LIN {X -127.4222,Y -50.5448,Z 181,A -155.3504,B 4.9597,C 0.2907,E1 4.8193,E2 248.002} C_DIS
LIN {X -128.4048,Y -47.9879,Z 181,A -156.9289,B 4.9597,C 0.2911,E1 4.8177,E2 249.6345} C_DIS
LIN {X -129.6974,Y -44.3795,Z 181,A -158.3245,B 4.9601,C 0.2852,E1 4.8165,E2 251.0033} C_DIS
LIN {X -131.1227,Y -39.9689,Z 181,A -160.1788,B 4.9604,C 0.2794,E1 4.8149,E2 252.846} C_DIS
LIN {X -132.6137,Y -34.708,Z 181,A -162.7791,B 4.9606,C 0.2756,E1 4.813,E2 255.4845} C_DIS
LIN {X -133.7601,Y -29.987,Z 181,A -164.6322,B 4.961,C 0.2687,E1 4.8118,E2 257.3141} C_DIS
LIN {X -134.5901,Y -26.0051,Z 181,A -166.4043,B 4.9612,C 0.2645,E1 4.8108,E2 259.0942} C_DIS
LIN {X -135.2142,Y -22.535,Z 181,A -167.8736,B 4.9614,C 0.2604,E1 4.8101,E2 260.5619} C_DIS
LIN {X -135.7342,Y -19.1571,Z 181,A -169.4073,B 4.9616,C 0.2572,E1 4.8095,E2 262.1079} C_DIS
LIN {X -136.1691,Y -15.7773,Z 181,A -170.7766,B 4.9618,C 0.2527,E1 4.8091,E2 263.4693} C_DIS
LIN {X -136.5191,Y -12.4002,Z 181,A -172.4163,B 4.9619,C 0.2504,E1 4.8086,E2 265.1357} C_DIS
LIN {X -136.8218,Y -8.399,Z 181,A -174.0209,B 4.9622,C 0.2451,E1 4.8083,E2 266.73} C_DIS
LIN {X -137.0078,Y -4.482,Z 181,A -175.6326,B 4.9624,C 0.2403,E1 4.8081,E2 268.3372} C_DIS
LIN {X -137.0637,Y -2.0849,Z 181,A -176.846,B 4.9624,C 0.239,E1 4.8081,E2 269.5761} C_DIS
LIN {X -137.0619,Y 2.1912,Z 181,A -178.5932,B 4.9628,C 0.2337,E1 4.8081,E2 271.317} C_DIS
LIN {X -136.938,Y 6.2553,Z 181,A 179.5206,B 4.9629,C 0.2303,E1 4.8083,E2 273.2253} C_DIS
LIN {X -136.6544,Y 10.81,Z 181,A 177.7567,B 4.9632,C 0.2238,E1 4.8086,E2 274.9699} C_DIS
LIN {X -136.4364,Y 13.2611,Z 181,A 176.6099,B 4.9632,C 0.2217,E1 4.8089,E2 276.1305} C_DIS
LIN {X -135.9488,Y 17.5695,Z 181,A 174.7524,B 4.9635,C 0.217,E1 4.8096,E2 277.9922} C_DIS
LIN {X -135.4593,Y 21.0118,Z 181,A 173.2902,B 4.9637,C 0.2129,E1 4.8101,E2 279.4544} C_DIS
LIN {X -134.8751,Y 24.4851,Z 181,A 171.6938,B 4.9638,C 0.2098,E1 4.8109,E2 281.065} C_DIS
LIN {X -134.1824,Y 28.0407,Z 181,A 170.242,B 4.964,C 0.2051,E1 4.8117,E2 282.5079} C_DIS
LIN {X -133.5527,Y 30.8949,Z 181,A 169.017,B 4.9642,C 0.2017,E1 4.8125,E2 283.7323} C_DIS
LIN {X -132.8302,Y 33.8649,Z 181,A 167.5658,B 4.9642,C 0.1995,E1 4.8135,E2 285.2039} C_DIS
LIN {X -131.1613,Y 39.8428,Z 181,A 165.1863,B 4.9646,C 0.1908,E1 4.8153,E2 287.5547} C_DIS
LIN {X -130.1059,Y 43.1639,Z 181,A 162.9954,B 4.9646,C 0.1925,E1 4.8173,E2 289.8349} C_DIS
LIN {X -128.6823,Y 47.2456,Z 181,A 161.6199,B 4.9648,C 0.1843,E1 4.8185,E2 291.156} C_DIS
LIN {X -127.3812,Y 50.6465,Z 181,A 160.1255,B 4.965,C 0.1801,E1 4.82,E2 292.6456} C_DIS
LIN {X -126.3636,Y 53.1315,Z 181,A 158.9035,B 4.965,C 0.1779,E1 4.8213,E2 293.879} C_DIS
LIN {X -125.0269,Y 56.2046,Z 181,A 157.4516,B 4.9652,C 0.1747,E1 4.823,E2 295.336} C_DIS
LIN {X -123.2922,Y 59.9191,Z 181,A 155.3859,B 4.9652,C 0.173,E1 4.8255,E2 297.4435} C_DIS
LIN {X -121.8194,Y 62.8584,Z 181,A 154.3358,B 4.9654,C 0.167,E1 4.8268,E2 298.4527} C_DIS
LIN {X -119.3576,Y 67.4167,Z 181,A 151.941,B 4.9656,C 0.1634,E1 4.83,E2 300.8739} C_DIS
LIN {X -117.0745,Y 71.3086,Z 181,A 149.9679,B 4.9656,C 0.1596,E1 4.8329,E2 302.856} C_DIS
LIN {X -114.569,Y 75.267,Z 181,A 148.1433,B 4.9659,C 0.1538,E1 4.8356,E2 304.6626} C_DIS
LIN {X -112.3179,Y 78.5874,Z 181,A 146.2806,B 4.9659,C 0.1514,E1 4.8386,E2 306.5466} C_DIS
LIN {X -109.7242,Y 82.17,Z 181,A 144.459,B 4.9661,C 0.147,E1 4.8416,E2 308.3633} C_DIS
LIN {X -107.0972,Y 85.5653,Z 181,A 142.5826,B 4.9661,C 0.1436,E1 4.8448,E2 310.2483} C_DIS
LIN {X -104.1716,Y 89.1045,Z 181,A 140.6095,B 4.9663,C 0.1399,E1 4.8484,E2 312.2263} C_DIS
LIN {X -101.272,Y 92.3865,Z 181,A 138.7169,B 4.9663,C 0.1366,E1 4.8519,E2 314.1249} C_DIS
LIN {X -98.1456,Y 95.7013,Z 181,A 136.7588,B 4.9665,C 0.1332,E1 4.8557,E2 316.088} C_DIS
LIN {X -94.866,Y 98.9527,Z 181,A 134.8418,B 4.9665,C 0.1293,E1 4.8596,E2 318.0018} C_DIS
LIN {X -91.7482,Y 101.8508,Z 181,A 133.0898,B 4.9667,C 0.1257,E1 4.8632,E2 319.749} C_DIS
LIN {X -88.6582,Y 104.5509,Z 181,A 131.2714,B 4.9667,C 0.1234,E1 4.867,E2 321.5786} C_DIS
LIN {X -85.1052,Y 107.4634,Z 181,A 129.2973,B 4.9667,C 0.1205,E1 4.8713,E2 323.5576} C_DIS
LIN {X -81.5224,Y 110.2063,Z 181,A 127.3566,B 4.9668,C 0.1178,E1 4.8757,E2 325.5035} C_DIS
LIN {X -77.8059,Y 112.8604,Z 181,A 125.4575,B 4.9669,C 0.1147,E1 4.88,E2 327.3999} C_DIS
LIN {X -74.2399,Y 115.2378,Z 181,A 123.4719,B 4.9669,C 0.1137,E1 4.8847,E2 329.4078} C_DIS
LIN {X -70.0881,Y 117.8085,Z 181,A 121.5767,B 4.967,C 0.1094,E1 4.8892,E2 331.2837} C_DIS
LIN {X -66.2568,Y 120.0051,Z 181,A 119.7445,B 4.967,C 0.1068,E1 4.8936,E2 333.1129} C_DIS
LIN {X -63.4029,Y 121.5352,Z 181,A 118.4017,B 4.9671,C 0.1049,E1 4.8969,E2 334.4533} C_DIS
LIN {X -59.8434,Y 123.3291,Z 181,A 116.7251,B 4.9671,C 0.103,E1 4.9011,E2 336.1302} C_DIS
LIN {X -57.2193,Y 124.566,Z 181,A 115.455,B 4.9671,C 0.1021,E1 4.9044,E2 337.4063} C_DIS
LIN {X -51.8982,Y 126.8767,Z 181,A 113.0963,B 4.9673,C 0.0989,E1 4.9104,E2 339.7554} C_DIS
LIN {X -47.8825,Y 128.4443,Z 181,A 110.7307,B 4.9672,C 0.1025,E1 4.9168,E2 342.1878} C_DIS
LIN {X -43.7874,Y 129.8983,Z 181,A 109.5162,B 4.9673,C 0.0951,E1 4.9198,E2 343.3284} C_DIS
LIN {X -39.1295,Y 131.3771,Z 181,A 107.4064,B 4.9673,C 0.0942,E1 4.9254,E2 345.4452} C_DIS
LIN {X -35.3632,Y 132.4391,Z 181,A 105.689,B 4.9673,C 0.0938,E1 4.9301,E2 347.1714} C_DIS
LIN {X -31.993,Y 133.2934,Z 181,A 104.1859,B 4.9673,C 0.0934,E1 4.9342,E2 348.6797} C_DIS
LIN {X -28.5696,Y 134.0694,Z 181,A 102.7942,B 4.9673,C 0.0918,E1 4.9379,E2 350.0614} C_DIS
LIN {X -25.5519,Y 134.6767,Z 181,A 101.3842,B 4.9673,C 0.0924,E1 4.9418,E2 351.4857} C_DIS
LIN {X -21.9917,Y 135.3048,Z 181,A 99.9775,B 4.9674,C 0.0907,E1 4.9457,E2 352.8789} C_DIS
LIN {X -19.0809,Y 135.7451,Z 181,A 98.656,B 4.9674,C 0.0912,E1 4.9494,E2 354.2107} C_DIS
LIN {X -11.6638,Y 136.5822,Z 181,A 95.8359,B 4.9674,C 0.0873,E1 4.9571,E2 356.9929} C_DIS
LIN {X -8.5421,Y 136.813,Z 181,A 94.3095,B 4.9674,C 0.0894,E1 4.9614,E2 358.5452} C_DIS
LIN {X -4.7604,Y 136.9979,Z 181,A 92.5308,B 4.9674,C 0.0913,E1 4.9664,E2 360.347} C_DIS
LIN {X 0.0145,Y 137.0815,Z 181,A 90.5073,B 4.9674,C 0.0917,E1 4.9721,E2 362.373} C_DIS
LIN {X 4.3871,Y 137.0104,Z 181,A 88.3455,B 4.9674,C 0.0955,E1 4.9783,E2 364.5743} C_DIS
LIN {X 8.7391,Y 136.8008,Z 181,A 86.9314,B 4.9674,C 0.0915,E1 4.9821,E2 365.9385} C_DIS
LIN {X 18.6225,Y 135.8104,Z 181,A 82.9311,B 4.9674,C 0.0913,E1 4.9931,E2 369.9192} C_DIS
LIN {X 22.8115,Y 135.168,Z 181,A 81.1423,B 4.9674,C 0.0924,E1 4.998,E2 371.7095} C_DIS
LIN {X 26.6873,Y 134.4578,Z 181,A 79.567,B 4.9674,C 0.0925,E1 5.0023,E2 373.2756} C_DIS
LIN {X 29.3272,Y 133.9058,Z 181,A 78.423,B 4.9674,C 0.0934,E1 5.0055,E2 374.4213} C_DIS
LIN {X 32.1885,Y 133.2463,Z 181,A 77.1384,B 4.9674,C 0.0949,E1 5.009,E2 375.7125} C_DIS
LIN {X 35.9507,Y 132.2824,Z 181,A 75.4086,B 4.9673,C 0.0974,E1 5.0137,E2 377.455} C_DIS
LIN {X 40.4649,Y 130.9709,Z 181,A 73.532,B 4.9673,C 0.0981,E1 5.0187,E2 379.3204} C_DIS
LIN {X 43.7971,Y 129.8951,Z 181,A 72.1572,B 4.9673,C 0.0984,E1 5.0223,E2 380.684} C_DIS
LIN {X 47.5976,Y 128.551,Z 181,A 70.598,B 4.9673,C 0.0986,E1 5.0264,E2 382.2277} C_DIS
LIN {X 50.1867,Y 127.5626,Z 181,A 69.3569,B 4.9673,C 0.1009,E1 5.0296,E2 383.4787} C_DIS
LIN {X 52.8036,Y 126.5006,Z 181,A 68.1774,B 4.9672,C 0.1022,E1 5.0327,E2 384.6578} C_DIS
LIN {X 55.9354,Y 125.1473,Z 181,A 66.7595,B 4.9672,C 0.1038,E1 5.0363,E2 386.0746} C_DIS
LIN {X 59.3192,Y 123.5795,Z 181,A 65.1645,B 4.9672,C 0.1061,E1 5.0403,E2 387.6739} C_DIS
LIN {X 62.7355,Y 121.882,Z 181,A 63.5393,B 4.9671,C 0.1086,E1 5.0444,E2 389.3028} C_DIS
LIN {X 66.8274,Y 119.6888,Z 181,A 61.615,B 4.967,C 0.1112,E1 5.0491,E2 391.2251} C_DIS
LIN {X 70.7239,Y 117.4281,Z 181,A 59.7788,B 4.967,C 0.1134,E1 5.0535,E2 393.0556} C_DIS
LIN {X 74.399,Y 115.1348,Z 181,A 57.9788,B 4.9669,C 0.116,E1 5.0577,E2 394.8543} C_DIS
LIN {X 78.0937,Y 112.6614,Z 181,A 56.1818,B 4.9669,C 0.1183,E1 5.0619,E2 396.6439} C_DIS
LIN {X 81.4416,Y 110.2658,Z 181,A 54.4735,B 4.9668,C 0.1211,E1 5.0657,E2 398.3508} C_DIS
LIN {X 84.9148,Y 107.6138,Z 181,A 52.828,B 4.9668,C 0.122,E1 5.0693,E2 399.9742} C_DIS
LIN {X 87.9841,Y 105.1189,Z 181,A 51.0867,B 4.9666,C 0.1262,E1 5.0731,E2 401.7266} C_DIS
LIN {X 91.2872,Y 102.2636,Z 181,A 49.2845,B 4.9666,C 0.1293,E1 5.0769,E2 403.5262} C_DIS
LIN {X 95.01,Y 98.8151,Z 181,A 47.4254,B 4.9666,C 0.1301,E1 5.0806,E2 405.3535} C_DIS
LIN {X 97.4012,Y 96.4584,Z 181,A 45.8405,B 4.9664,C 0.1353,E1 5.0838,E2 406.9611} C_DIS
LIN {X 100.7401,Y 92.9659,Z 181,A 44.0324,B 4.9664,C 0.1368,E1 5.0872,E2 408.7435} C_DIS
LIN {X 103.0225,Y 90.4306,Z 181,A 42.4295,B 4.9662,C 0.1422,E1 5.0902,E2 410.3686} C_DIS
LIN {X 106.0826,Y 86.8197,Z 181,A 40.5868,B 4.9662,C 0.1447,E1 5.0935,E2 412.1952} C_DIS
LIN {X 108.6774,Y 83.5493,Z 181,A 38.776,B 4.966,C 0.1495,E1 5.0966,E2 414.0146} C_DIS
LIN {X 111.4246,Y 79.8482,Z 181,A 36.9393,B 4.9659,C 0.1528,E1 5.0996,E2 415.8408} C_DIS
LIN {X 113.8804,Y 76.3051,Z 181,A 35.2325,B 4.9659,C 0.1557,E1 5.1023,E2 417.5365} C_DIS
LIN {X 116.1332,Y 72.8313,Z 181,A 33.4741,B 4.9657,C 0.1603,E1 5.1049,E2 419.2991} C_DIS
LIN {X 118.3907,Y 69.1009,Z 181,A 31.7162,B 4.9655,C 0.1639,E1 5.1074,E2 421.0496} C_DIS
LIN {X 120.5422,Y 65.2758,Z 181,A 29.8915,B 4.9654,C 0.1683,E1 5.1099,E2 422.874} C_DIS
LIN {X 122.3185,Y 61.8781,Z 181,A 28.4935,B 4.9654,C 0.1696,E1 5.1117,E2 424.2472} C_DIS
LIN {X 123.9901,Y 58.4599,Z 181,A 26.9069,B 4.9652,C 0.1736,E1 5.1136,E2 425.8341} C_DIS
LIN {X 125.4874,Y 55.1746,Z 181,A 25.2581,B 4.965,C 0.1794,E1 5.1155,E2 427.5011} C_DIS
LIN {X 126.8213,Y 52.0353,Z 181,A 24.0296,B 4.965,C 0.1805,E1 5.1168,E2 428.7058} C_DIS
LIN {X 127.9651,Y 49.1514,Z 181,A 22.8027,B 4.9649,C 0.183,E1 5.118,E2 429.9245} C_DIS
LIN {X 129.1015,Y 46.0828,Z 181,A 21.4926,B 4.9648,C 0.1858,E1 5.1193,E2 431.2282} C_DIS
LIN {X 130.0263,Y 43.4028,Z 181,A 20.2799,B 4.9646,C 0.1894,E1 5.1204,E2 432.445} C_DIS
LIN {X 131.1082,Y 40.0163,Z 181,A 18.834,B 4.9646,C 0.1929,E1 5.1216,E2 433.8866} C_DIS
LIN {X 132.0676,Y 36.7268,Z 181,A 17.428,B 4.9644,C 0.1964,E1 5.1226,E2 435.2903} C_DIS
LIN {X 133.0944,Y 32.8188,Z 181,A 15.856,B 4.9642,C 0.1994,E1 5.1237,E2 436.8487} C_DIS
LIN {X 133.6857,Y 30.3126,Z 181,A 14.8245,B 4.9642,C 0.2018,E1 5.1244,E2 437.8752} C_DIS
LIN {X 134.3424,Y 27.2545,Z 181,A 13.4894,B 4.964,C 0.2058,E1 5.1251,E2 439.2145} C_DIS
LIN {X 134.9912,Y 23.8366,Z 181,A 11.9946,B 4.9638,C 0.2104,E1 5.1259,E2 440.7154} C_DIS
LIN {X 135.5678,Y 20.3107,Z 181,A 10.6544,B 4.9638,C 0.2125,E1 5.1265,E2 442.0375} C_DIS
LIN {X 135.9236,Y 17.7618,Z 181,A 9.048,B 4.9632,C 0.2229,E1 5.1271,E2 443.711} C_DIS
LIN {X 136.4483,Y 13.1377,Z 181,A 7.6818,B 4.9634,C 0.2203,E1 5.1274,E2 445.006} C_DIS
LIN {X 136.8955,Y 7.1008,Z 181,A 5.121,B 4.963,C 0.228,E1 5.1279,E2 447.5724} C_DIS
LIN {X 137.0396,Y 3.3361,Z 181,A 2.9853,B 4.9624,C 0.2403,E1 5.1281,E2 449.7797} C_DIS
LIN {X 137.0602,Y -2.2939,Z 181,A 1.7231,B 4.9628,C 0.2317,E1 5.1281,E2 450.9063} C_DIS
LIN {X 136.8901,Y -7.2074,Z 181,A -0.651,B 4.9624,C 0.242,E1 5.1278,E2 453.3225} C_DIS
LIN {X 136.2682,Y -14.8915,Z 181,A -3.7237,B 4.962,C 0.2491,E1 5.127,E2 456.3787} C_DIS
LIN {X 135.7302,Y -19.1848,Z 181,A -5.7946,B 4.9616,C 0.2579,E1 5.1262,E2 458.4843} C_DIS
LIN {X 135.2011,Y -22.6135,Z 181,A -7.1721,B 4.9614,C 0.2609,E1 5.1256,E2 459.8538} C_DIS
LIN {X 134.6162,Y -25.8687,Z 181,A -8.1979,B 4.9614,C 0.2598,E1 5.1251,E2 460.8355} C_DIS
LIN {X 133.9971,Y -28.9045,Z 181,A -9.4926,B 4.9613,C 0.2634,E1 5.1244,E2 462.1313} C_DIS
LIN {X 133.233,Y -32.2435,Z 181,A -10.8818,B 4.9611,C 0.2668,E1 5.1235,E2 463.5162} C_DIS
LIN {X 132.3618,Y -35.6532,Z 181,A -12.2736,B 4.9609,C 0.2697,E1 5.1225,E2 464.8991} C_DIS
LIN {X 131.6135,Y -38.322,Z 181,A -13.3402,B 4.9609,C 0.2716,E1 5.1217,E2 465.955} C_DIS
LIN {X 130.7283,Y -41.243,Z 181,A -14.7978,B 4.9605,C 0.2777,E1 5.1205,E2 467.4369} C_DIS
LIN {X 129.5874,Y -44.6965,Z 181,A -16.2283,B 4.9603,C 0.2806,E1 5.1192,E2 468.8572} C_DIS
LIN {X 128.2347,Y -48.4421,Z 181,A -17.84,B 4.9601,C 0.2843,E1 5.1176,E2 470.4636} C_DIS
LIN {X 126.9922,Y -51.6117,Z 181,A -19.2168,B 4.9599,C 0.2874,E1 5.1162,E2 471.8358} C_DIS
LIN {X 125.5455,Y -55.0403,Z 181,A -20.8621,B 4.9596,C 0.2928,E1 5.1144,E2 473.4939} C_DIS
LIN {X 123.4346,Y -59.6225,Z 181,A -22.7964,B 4.9594,C 0.2959,E1 5.1121,E2 475.4077} C_DIS
LIN {X 120.8614,Y -64.6819,Z 181,A -25.1445,B 4.9591,C 0.3016,E1 5.1091,E2 477.7548} C_DIS
LIN {X 118.6742,Y -68.612,Z 181,A -26.9437,B 4.9589,C 0.3052,E1 5.1066,E2 479.5453} C_DIS
LIN {X 116.503,Y -72.2375,Z 181,A -28.697,B 4.9586,C 0.3094,E1 5.1041,E2 481.2985} C_DIS
LIN {X 114.0621,Y -76.0329,Z 181,A -30.5338,B 4.9584,C 0.3133,E1 5.1013,E2 483.1307} C_DIS
LIN {X 111.5188,Y -79.7164,Z 181,A -32.3333,B 4.9582,C 0.3168,E1 5.0984,E2 484.9226} C_DIS
LIN {X 108.9758,Y -83.1592,Z 181,A -34.108,B 4.9579,C 0.3208,E1 5.0954,E2 486.6971} C_DIS
LIN {X 106.1641,Y -86.7198,Z 181,A -35.9666,B 4.9577,C 0.3246,E1 5.0922,E2 488.5525} C_DIS
LIN {X 103.2841,Y -90.1307,Z 181,A -38.5687,B 4.9567,C 0.3386,E1 5.0872,E2 491.2503} C_DIS
LIN {X 98.8406,Y -94.9831,Z 181,A -40.4642,B 4.9571,C 0.333,E1 5.0838,E2 493.0389} C_DIS
LIN {X 95.6206,Y -98.224,Z 181,A -42.8084,B 4.9564,C 0.3428,E1 5.079,E2 495.4406} C_DIS
LIN {X 92.1511,Y -101.4857,Z 181,A -44.6325,B 4.9564,C 0.3445,E1 5.0753,E2 497.245} C_DIS
LIN {X 89.0614,Y -104.2082,Z 181,A -45.9165,B 4.9564,C 0.3421,E1 5.0727,E2 498.4743} C_DIS
LIN {X 85.8115,Y -106.9001,Z 181,A -47.7116,B 4.9562,C 0.3458,E1 5.0688,E2 500.2748} C_DIS
LIN {X 82.4043,Y -109.5479,Z 181,A -49.4965,B 4.956,C 0.3488,E1 5.0648,E2 502.0588} C_DIS
LIN {X 79.4611,Y -111.7014,Z 181,A -50.8313,B 4.956,C 0.349,E1 5.0619,E2 503.3703} C_DIS
LIN {X 76.484,Y -113.7609,Z 181,A -52.5018,B 4.9557,C 0.3537,E1 5.058,E2 505.0624} C_DIS
LIN {X 72.6713,Y -116.233,Z 181,A -54.3702,B 4.9555,C 0.3563,E1 5.0536,E2 506.9283} C_DIS
LIN {X 68.7676,Y -118.5841,Z 181,A -56.1804,B 4.9554,C 0.3581,E1 5.0492,E2 508.7278} C_DIS
LIN {X 65.229,Y -120.5674,Z 181,A -57.924,B 4.9551,C 0.3612,E1 5.0449,E2 510.479} C_DIS
LIN {X 61.1245,Y -122.6975,Z 181,A -59.5909,B 4.9551,C 0.3605,E1 5.0409,E2 512.1128} C_DIS
LIN {X 58.5464,Y -123.9487,Z 181,A -61.3471,B 4.9545,C 0.3691,E1 5.0363,E2 513.9421} C_DIS
LIN {X 54.6931,Y -125.6956,Z 181,A -62.5684,B 4.9549,C 0.3645,E1 5.0333,E2 515.094} C_DIS
LIN {X 46.1668,Y -129.0712,Z 181,A -66.5389,B 4.9544,C 0.3706,E1 5.0229,E2 519.0852} C_DIS
LIN {X 42.7434,Y -130.2459,Z 181,A -67.8846,B 4.9544,C 0.3701,E1 5.0194,E2 520.4103} C_DIS
LIN {X 39.616,Y -131.2307,Z 181,A -69.2298,B 4.9544,C 0.3711,E1 5.0158,E2 521.7531} C_DIS
LIN {X 37.127,Y -131.9556,Z 181,A -70.4001,B 4.9542,C 0.3731,E1 5.0127,E2 522.9354} C_DIS
LIN {X 33.0424,Y -133.0389,Z 181,A -72.0524,B 4.9542,C 0.3732,E1 5.0082,E2 524.5741} C_DIS
LIN {X 30.3153,Y -133.6851,Z 181,A -73.2373,B 4.9542,C 0.3743,E1 5.005,E2 525.7614} C_DIS
LIN {X 26.8252,Y -134.4298,Z 181,A -74.6979,B 4.9542,C 0.375,E1 5.001,E2 527.2189} C_DIS
LIN {X 24.1857,Y -134.9287,Z 181,A -76.8599,B 4.9531,C 0.3879,E1 4.9947,E2 529.5155} C_DIS
LIN {X 16.9844,Y -136.0251,Z 181,A -78.839,B 4.9539,C 0.377,E1 4.9896,E2 531.3592} C_DIS
LIN {X 12.6189,Y -136.4981,Z 181,A -80.9968,B 4.9536,C 0.3815,E1 4.9835,E2 533.5598} C_DIS
LIN {X 9.2394,Y -136.7696,Z 181,A -82.4515,B 4.9536,C 0.3824,E1 4.9794,E2 535.0201} C_DIS
LIN {X 5.8129,Y -136.9569,Z 181,A -83.8434,B 4.9536,C 0.3823,E1 4.9755,E2 536.4072} C_DIS
LIN {X 2.5453,Y -137.056,Z 181,A -84.6933,B 4.954,C 0.3767,E1 4.9733,E2 537.1908} C_DIS
LIN {X 2.5453,Y -137.056,Z 181,A -84.6933,B 4.954,C 0.3767,E1 4.9733,E2 537.1908} C_DIS
Enddeposition()
LIN {X 0.9801,Y -137.9766,Z 181,A -85.0091,B 4.9146,C 0.3749,E1 4.933,E2 537.5057} C_DIS
Startdeposition()
$VEL.CP = VEL_PRINT
LIN {X 4.6039,Y -137.9071,Z 181,A -83.4141,B 4.9146,C 0.3736,E1 4.9375,E2 535.8982} C_DIS
LIN {X 7.7048,Y -137.7686,Z 181,A -82.0968,B 4.9147,C 0.3729,E1 4.9412,E2 534.5765} C_DIS
LIN {X 10.9129,Y -137.5512,Z 181,A -80.8244,B 4.9147,C 0.3732,E1 4.9447,E2 533.3117} C_DIS
LIN {X 14.4702,Y -137.2211,Z 181,A -79.3015,B 4.9147,C 0.3721,E1 4.949,E2 531.7828} C_DIS
LIN {X 18.7238,Y -136.7076,Z 181,A -77.5399,B 4.9148,C 0.3715,E1 4.9538,E2 530.0225} C_DIS
LIN {X 22.2329,Y -136.1794,Z 181,A -76.192,B 4.9148,C 0.3721,E1 4.9575,E2 528.6903} C_DIS
LIN {X 25.108,Y -135.6803,Z 181,A -74.8358,B 4.915,C 0.3696,E1 4.9613,E2 527.3144} C_DIS
LIN {X 28.8616,Y -134.9295,Z 181,A -73.302,B 4.915,C 0.3692,E1 4.9655,E2 525.7869} C_DIS
LIN {X 31.6997,Y -134.2923,Z 181,A -72.1492,B 4.915,C 0.369,E1 4.9686,E2 524.6406} C_DIS
LIN {X 34.8347,Y -133.5139,Z 181,A -70.7533,B 4.9152,C 0.3672,E1 4.9724,E2 523.2367} C_DIS
LIN {X 38.0538,Y -132.6323,Z 181,A -69.3785,B 4.9152,C 0.3661,E1 4.9761,E2 521.8624} C_DIS
LIN {X 41.7013,Y -131.5293,Z 181,A -67.9232,B 4.9152,C 0.3661,E1 4.9799,E2 520.4229} C_DIS
LIN {X 44.3961,Y -130.6466,Z 181,A -66.6424,B 4.9154,C 0.3637,E1 4.9834,E2 519.1276} C_DIS
LIN {X 47.5995,Y -129.5139,Z 181,A -65.2454,B 4.9155,C 0.3623,E1 4.987,E2 517.7315} C_DIS
LIN {X 50.7912,Y -128.2958,Z 181,A -63.7183,B 4.9157,C 0.3593,E1 4.9911,E2 516.1891} C_DIS
LIN {X 54.4474,Y -126.7849,Z 181,A -62.2039,B 4.9157,C 0.3589,E1 4.9949,E2 514.6904} C_DIS
LIN {X 57.2108,Y -125.5641,Z 181,A -60.9781,B 4.9159,C 0.3577,E1 4.998,E2 513.4674} C_DIS
LIN {X 60.347,Y -124.0872,Z 181,A -59.5906,B 4.9159,C 0.3564,E1 5.0015,E2 512.0857} C_DIS
LIN {X 63.3753,Y -122.5689,Z 181,A -58.0603,B 4.9162,C 0.3529,E1 5.0054,E2 510.538} C_DIS
LIN {X 67.266,Y -120.4774,Z 181,A -56.373,B 4.9162,C 0.3521,E1 5.0095,E2 508.8688} C_DIS
LIN {X 70.2684,Y -118.7515,Z 181,A -54.9436,B 4.9164,C 0.35,E1 5.0129,E2 507.4394} C_DIS
LIN {X 73.3161,Y -116.8943,Z 181,A -53.3895,B 4.9166,C 0.3467,E1 5.0166,E2 505.8746} C_DIS
LIN {X 76.98,Y -114.5148,Z 181,A -51.6286,B 4.9168,C 0.3444,E1 5.0207,E2 504.1193} C_DIS
LIN {X 80.6162,Y -111.9848,Z 181,A -49.8411,B 4.917,C 0.3419,E1 5.0248,E2 502.3372} C_DIS
LIN {X 83.4723,Y -109.8724,Z 181,A -48.4303,B 4.9171,C 0.3401,E1 5.0279,E2 500.9336} C_DIS
LIN {X 86.2779,Y -107.6833,Z 181,A -46.94,B 4.9173,C 0.3372,E1 5.0312,E2 499.4405} C_DIS
LIN {X 89.0299,Y -105.4193,Z 181,A -45.5406,B 4.9174,C 0.3354,E1 5.0342,E2 498.0504} C_DIS
LIN {X 91.7612,Y -103.0505,Z 181,A -44.0812,B 4.9176,C 0.3331,E1 5.0372,E2 496.5952} C_DIS
LIN {X 94.3966,Y -100.642,Z 181,A -42.6286,B 4.9178,C 0.3305,E1 5.0402,E2 495.1453} C_DIS
LIN {X 97.337,Y -97.8002,Z 181,A -40.8978,B 4.918,C 0.3265,E1 5.0436,E2 493.4087} C_DIS
LIN {X 100.336,Y -94.7209,Z 181,A -39.1333,B 4.9182,C 0.323,E1 5.0471,E2 491.6454} C_DIS
LIN {X 103.1142,Y -91.6896,Z 181,A -37.5493,B 4.9184,C 0.321,E1 5.05,E2 490.0761} C_DIS
LIN {X 105.4501,Y -88.9933,Z 181,A -35.973,B 4.9187,C 0.3164,E1 5.0529,E2 488.4861} C_DIS
LIN {X 108.2377,Y -85.5814,Z 181,A -34.2888,B 4.9188,C 0.3142,E1 5.0558,E2 486.8194} C_DIS
LIN {X 110.4077,Y -82.7629,Z 181,A -32.8592,B 4.919,C 0.3115,E1 5.0582,E2 485.3947} C_DIS
LIN {X 112.5007,Y -79.8947,Z 181,A -31.4082,B 4.9192,C 0.3083,E1 5.0606,E2 483.9454} C_DIS
LIN {X 114.7962,Y -76.5584,Z 181,A -29.7289,B 4.9194,C 0.3043,E1 5.0632,E2 482.2649} C_DIS
LIN {X 117.0033,Y -73.1415,Z 181,A -28.1617,B 4.9196,C 0.3019,E1 5.0655,E2 480.7122} C_DIS
LIN {X 118.7753,Y -70.2278,Z 181,A -26.6687,B 4.9199,C 0.2973,E1 5.0677,E2 479.2079} C_DIS
LIN {X 120.9472,Y -66.4176,Z 181,A -24.9601,B 4.92,C 0.2943,E1 5.07,E2 477.5125} C_DIS
LIN {X 122.6113,Y -63.2919,Z 181,A -23.5819,B 4.9202,C 0.2918,E1 5.0718,E2 476.145} C_DIS
LIN {X 124.1285,Y -60.2633,Z 181,A -22.1794,B 4.9204,C 0.2882,E1 5.0735,E2 474.7419} C_DIS
LIN {X 125.6031,Y -57.1264,Z 181,A -20.6382,B 4.9207,C 0.283,E1 5.0753,E2 473.1861} C_DIS
LIN {X 127.0278,Y -53.8827,Z 181,A -19.3485,B 4.9207,C 0.2817,E1 5.0767,E2 471.9188} C_DIS
LIN {X 128.3291,Y -50.7056,Z 181,A -17.9625,B 4.921,C 0.2784,E1 5.0781,E2 470.5368} C_DIS
LIN {X 129.5449,Y -47.5135,Z 181,A -16.5838,B 4.9211,C 0.2752,E1 5.0795,E2 469.162} C_DIS
LIN {X 130.6753,Y -44.31,Z 181,A -15.2456,B 4.9213,C 0.2724,E1 5.0807,E2 467.832} C_DIS
LIN {X 131.6944,Y -41.1844,Z 181,A -13.8873,B 4.9215,C 0.2688,E1 5.0819,E2 466.4735} C_DIS
LIN {X 132.6576,Y -37.9674,Z 181,A -12.533,B 4.9217,C 0.2655,E1 5.0829,E2 465.1232} C_DIS
LIN {X 133.5589,Y -34.6619,Z 181,A -11.0655,B 4.9219,C 0.2609,E1 5.084,E2 463.6487} C_DIS
LIN {X 134.4183,Y -31.1575,Z 181,A -9.6758,B 4.9221,C 0.2583,E1 5.0849,E2 462.2718} C_DIS
LIN {X 135.1425,Y -27.848,Z 181,A -8.4602,B 4.9221,C 0.2571,E1 5.0856,E2 461.0799} C_DIS
LIN {X 135.6957,Y -25.022,Z 181,A -7.1712,B 4.9224,C 0.2524,E1 5.0862,E2 459.7779} C_DIS
LIN {X 136.2466,Y -21.8242,Z 181,A -5.8641,B 4.9225,C 0.2492,E1 5.0868,E2 458.4749} C_DIS
LIN {X 136.7188,Y -18.6385,Z 181,A -4.4356,B 4.9228,C 0.2441,E1 5.0874,E2 457.0335} C_DIS
LIN {X 137.1138,Y -15.4677,Z 181,A -3.2795,B 4.9228,C 0.2428,E1 5.0878,E2 455.8984} C_DIS
LIN {X 137.4258,Y -12.3985,Z 181,A -2.0368,B 4.923,C 0.2397,E1 5.0881,E2 454.6597} C_DIS
LIN {X 137.6777,Y -9.1803,Z 181,A -0.7373,B 4.9232,C 0.2365,E1 5.0883,E2 453.3645} C_DIS
LIN {X 137.85,Y -6.0683,Z 181,A 0.645,B 4.9234,C 0.2316,E1 5.0885,E2 451.9698} C_DIS
LIN {X 137.9741,Y -1.6104,Z 181,A 2.3233,B 4.9235,C 0.2288,E1 5.0886,E2 450.3125} C_DIS
LIN {X 137.9741,Y 1.6104,Z 181,A 3.5846,B 4.9236,C 0.226,E1 5.0886,E2 449.06} C_DIS
LIN {X 137.9071,Y 4.6039,Z 181,A 4.8245,B 4.9238,C 0.2225,E1 5.0886,E2 447.8197} C_DIS
LIN {X 137.7686,Y 7.7048,Z 181,A 6.108,B 4.924,C 0.219,E1 5.0883,E2 446.536} C_DIS
LIN {X 137.5121,Y 11.3762,Z 181,A 7.3704,B 4.924,C 0.2184,E1 5.0881,E2 445.3065} C_DIS
LIN {X 137.2746,Y 13.9732,Z 181,A 8.6501,B 4.9242,C 0.2125,E1 5.0877,E2 444.0009} C_DIS
LIN {X 136.9157,Y 17.1361,Z 181,A 9.9079,B 4.9244,C 0.2097,E1 5.0873,E2 442.7504} C_DIS
LIN {X 136.4802,Y 20.3151,Z 181,A 11.2053,B 4.9245,C 0.2065,E1 5.0868,E2 441.4566} C_DIS
LIN {X 135.9668,Y 23.5075,Z 181,A 12.6552,B 4.9247,C 0.2012,E1 5.0861,E2 439.9921} C_DIS
LIN {X 135.3564,Y 26.797,Z 181,A 13.8649,B 4.9247,C 0.1999,E1 5.0855,E2 438.8045} C_DIS
LIN {X 134.6808,Y 30.0085,Z 181,A 15.1604,B 4.9249,C 0.197,E1 5.0847,E2 437.5168} C_DIS
LIN {X 133.9454,Y 33.1389,Z 181,A 16.5225,B 4.9251,C 0.1929,E1 5.0838,E2 436.1505} C_DIS
LIN {X 133.0014,Y 36.7379,Z 181,A 17.9965,B 4.9251,C 0.1897,E1 5.0828,E2 434.6845} C_DIS
LIN {X 132.0741,Y 39.9438,Z 181,A 19.3665,B 4.9253,C 0.1861,E1 5.0817,E2 433.3157} C_DIS
LIN {X 131.0434,Y 43.2045,Z 181,A 20.7164,B 4.9254,C 0.1833,E1 5.0805,E2 431.9739} C_DIS
LIN {X 129.9299,Y 46.4456,Z 181,A 21.9466,B 4.9254,C 0.1821,E1 5.0794,E2 430.7675} C_DIS
LIN {X 128.9156,Y 49.197,Z 181,A 23.3034,B 4.9256,C 0.177,E1 5.0781,E2 429.3925} C_DIS
LIN {X 127.6547,Y 52.3816,Z 181,A 24.721,B 4.9258,C 0.1733,E1 5.0766,E2 427.9748} C_DIS
LIN {X 126.2705,Y 55.6343,Z 181,A 26.2348,B 4.9259,C 0.1688,E1 5.0749,E2 426.4543} C_DIS
LIN {X 124.8363,Y 58.7818,Z 181,A 27.5211,B 4.9259,C 0.1672,E1 5.0734,E2 425.1864} C_DIS
LIN {X 123.3593,Y 61.8226,Z 181,A 29.0146,B 4.9261,C 0.1624,E1 5.0715,E2 423.681} C_DIS
LIN {X 121.3436,Y 65.6908,Z 181,A 30.6694,B 4.9262,C 0.16,E1 5.0694,E2 422.0452} C_DIS
LIN {X 119.6364,Y 68.751,Z 181,A 32.0771,B 4.9263,C 0.157,E1 5.0675,E2 420.6428} C_DIS
LIN {X 117.8458,Y 71.7769,Z 181,A 33.5147,B 4.9264,C 0.1538,E1 5.0654,E2 419.2075} C_DIS
LIN {X 115.6064,Y 75.3299,Z 181,A 35.2302,B 4.9265,C 0.15,E1 5.0628,E2 417.495} C_DIS
LIN {X 113.5177,Y 78.4429,Z 181,A 36.7383,B 4.9266,C 0.1469,E1 5.0604,E2 415.9925} C_DIS
LIN {X 111.0892,Y 81.8449,Z 181,A 38.4954,B 4.9268,C 0.1426,E1 5.0576,E2 414.2321} C_DIS
LIN {X 108.7578,Y 84.9191,Z 181,A 39.9751,B 4.9268,C 0.1407,E1 5.0551,E2 412.7673} C_DIS
LIN {X 106.2677,Y 88.0144,Z 181,A 41.675,B 4.9269,C 0.1363,E1 5.052,E2 411.0606} C_DIS
LIN {X 103.3184,Y 91.4587,Z 181,A 43.4917,B 4.927,C 0.1331,E1 5.0487,E2 409.2518} C_DIS
LIN {X 100.642,Y 94.3966,Z 181,A 45.168,B 4.9271,C 0.1293,E1 5.0455,E2 407.5718} C_DIS
LIN {X 97.5226,Y 97.6159,Z 181,A 46.8772,B 4.9271,C 0.1275,E1 5.0422,E2 405.8814} C_DIS
LIN {X 95.0112,Y 100.0622,Z 181,A 48.3209,B 4.9272,C 0.1248,E1 5.0393,E2 404.4389} C_DIS
LIN {X 92.3902,Y 102.4871,Z 181,A 49.7743,B 4.9273,C 0.1223,E1 5.0363,E2 402.9889} C_DIS
LIN {X 89.3208,Y 105.1721,Z 181,A 51.4875,B 4.9273,C 0.1189,E1 5.0327,E2 401.273} C_DIS
LIN {X 85.7795,Y 108.0799,Z 181,A 53.3338,B 4.9275,C 0.1161,E1 5.0287,E2 399.4336} C_DIS
LIN {X 82.4519,Y 110.6393,Z 181,A 55.0767,B 4.9275,C 0.1131,E1 5.0248,E2 397.6905} C_DIS
LIN {X 79.1312,Y 113.0388,Z 181,A 56.6733,B 4.9275,C 0.1116,E1 5.0212,E2 396.107} C_DIS
LIN {X 76.2444,Y 115.0059,Z 181,A 58.0992,B 4.9276,C 0.1095,E1 5.0179,E2 394.6841} C_DIS
LIN {X 73.2315,Y 116.9472,Z 181,A 59.5598,B 4.9276,C 0.1076,E1 5.0145,E2 393.2269} C_DIS
LIN {X 70.2278,Y 118.7753,Z 181,A 60.9871,B 4.9276,C 0.1058,E1 5.0111,E2 391.8037} C_DIS
LIN {X 66.8589,Y 120.7032,Z 181,A 62.6695,B 4.9278,C 0.1026,E1 5.007,E2 390.1125} C_DIS
LIN {X 63.2919,Y 122.6113,Z 181,A 64.2687,B 4.9278,C 0.1013,E1 5.003,E2 388.5235} C_DIS
LIN {X 60.2633,Y 124.1285,Z 181,A 65.6289,B 4.9278,C 0.1001,E1 4.9996,E2 387.1692} C_DIS
LIN {X 57.1264,Y 125.6031,Z 181,A 67.1801,B 4.9278,C 0.0969,E1 4.9957,E2 385.6042} C_DIS
LIN {X 53.8827,Y 127.0278,Z 181,A 68.5007,B 4.9278,C 0.097,E1 4.9923,E2 384.3025} C_DIS
LIN {X 50.7056,Y 128.3291,Z 181,A 69.9086,B 4.9278,C 0.0957,E1 4.9887,E2 382.897} C_DIS
LIN {X 47.2903,Y 129.6254,Z 181,A 71.416,B 4.9279,C 0.0942,E1 4.9847,E2 381.3909} C_DIS
LIN {X 44.31,Y 130.6753,Z 181,A 72.672,B 4.9279,C 0.0936,E1 4.9814,E2 380.1422} C_DIS
LIN {X 41.1844,Y 131.6944,Z 181,A 74.0556,B 4.9279,C 0.0922,E1 4.9777,E2 378.7566} C_DIS
LIN {X 37.9674,Y 132.6576,Z 181,A 75.4361,B 4.9279,C 0.0911,E1 4.974,E2 377.3781} C_DIS
LIN {X 34.434,Y 133.6167,Z 181,A 76.986,B 4.928,C 0.0896,E1 4.9699,E2 375.8248} C_DIS
LIN {X 31.53,Y 134.3332,Z 181,A 78.1734,B 4.928,C 0.0894,E1 4.9666,E2 374.6446} C_DIS
LIN {X 28.3156,Y 135.0474,Z 181,A 79.5602,B 4.928,C 0.0883,E1 4.9629,E2 373.2558} C_DIS
LIN {X 25.022,Y 135.6957,Z 181,A 81.045,B 4.928,C 0.0864,E1 4.9587,E2 371.7601} C_DIS
LIN {X 21.6418,Y 136.2748,Z 181,A 82.2632,B 4.928,C 0.088,E1 4.9555,E2 370.5678} C_DIS
LIN {X 18.6385,Y 136.7188,Z 181,A 83.5483,B 4.928,C 0.0872,E1 4.9519,E2 369.2801} C_DIS
LIN {X 15.4677,Y 137.1138,Z 181,A 84.8989,B 4.928,C 0.0864,E1 4.9481,E2 367.927} C_DIS
LIN {X 12.3985,Y 137.4258,Z 181,A 86.3143,B 4.928,C 0.0845,E1 4.9442,E2 366.4954} C_DIS
LIN {X 9.1803,Y 137.6777,Z 181,A 87.5075,B 4.928,C 0.0858,E1 4.9409,E2 365.321} C_DIS
LIN {X 6.0683,Y 137.85,Z 181,A 88.7969,B 4.928,C 0.0856,E1 4.9373,E2 364.0327} C_DIS
LIN {X 3.0627,Y 137.9499,Z 181,A 90.0416,B 4.928,C 0.0855,E1 4.9338,E2 362.7891} C_DIS
LIN {X -0.082,Y 137.9835,Z 181,A 91.3457,B 4.928,C 0.0854,E1 4.9302,E2 361.4858} C_DIS
LIN {X -3.6178,Y 137.9345,Z 181,A 92.8346,B 4.928,C 0.0852,E1 4.926,E2 359.9949} C_DIS
LIN {X -7.7048,Y 137.7686,Z 181,A 94.5522,B 4.928,C 0.0852,E1 4.9212,E2 358.2758} C_DIS
LIN {X -10.9129,Y 137.5512,Z 181,A 95.8281,B 4.928,C 0.0859,E1 4.9177,E2 357.0079} C_DIS
LIN {X -13.9732,Y 137.2746,Z 181,A 97.171,B 4.928,C 0.0855,E1 4.9139,E2 355.6574} C_DIS
LIN {X -17.1361,Y 136.9157,Z 181,A 98.6199,B 4.928,C 0.0846,E1 4.9099,E2 354.1934} C_DIS
LIN {X -20.3151,Y 136.4802,Z 181,A 99.8088,B 4.928,C 0.0865,E1 4.9066,E2 353.023} C_DIS
LIN {X -23.5075,Y 135.9668,Z 181,A 101.1593,B 4.928,C 0.087,E1 4.9029,E2 351.6723} C_DIS
LIN {X -26.797,Y 135.3564,Z 181,A 102.5578,B 4.928,C 0.0876,E1 4.8991,E2 350.2734} C_DIS
LIN {X -30.0085,Y 134.6808,Z 181,A 103.9964,B 4.928,C 0.0876,E1 4.8951,E2 348.8262} C_DIS
LIN {X -33.4854,Y 133.8575,Z 181,A 105.4019,B 4.928,C 0.0893,E1 4.8913,E2 347.4313} C_DIS
LIN {X -36.4443,Y 133.0835,Z 181,A 106.7075,B 4.928,C 0.0898,E1 4.8878,E2 346.122} C_DIS
LIN {X -39.6627,Y 132.1601,Z 181,A 108.234,B 4.928,C 0.0895,E1 4.8837,E2 344.5795} C_DIS
LIN {X -43.3417,Y 130.9978,Z 181,A 109.5117,B 4.928,C 0.094,E1 4.8804,E2 343.3428} C_DIS
LIN {X -45.9991,Y 130.0909,Z 181,A 110.9066,B 4.928,C 0.0928,E1 4.8766,E2 341.9205} C_DIS
LIN {X -49.4285,Y 128.8256,Z 181,A 112.3488,B 4.928,C 0.095,E1 4.8729,E2 340.4887} C_DIS
LIN {X -52.3816,Y 127.6547,Z 181,A 113.8398,B 4.928,C 0.0947,E1 4.869,E2 338.9773} C_DIS
LIN {X -55.6343,Y 126.2705,Z 181,A 115.3539,B 4.9279,C 0.0959,E1 4.8651,E2 337.4585} C_DIS
LIN {X -58.7818,Y 124.8363,Z 181,A 116.7178,B 4.9279,C 0.0982,E1 4.8616,E2 336.1046} C_DIS
LIN {X -61.8226,Y 123.3593,Z 181,A 118.141,B 4.9279,C 0.0997,E1 4.8581,E2 334.6801} C_DIS
LIN {X -64.9208,Y 121.7573,Z 181,A 119.7082,B 4.9278,C 0.1005,E1 4.8542,E2 333.0991} C_DIS
LIN {X -68.751,Y 119.6364,Z 181,A 121.4554,B 4.9278,C 0.1036,E1 4.8499,E2 331.362} C_DIS
LIN {X -72.224,Y 117.5715,Z 181,A 123.2228,B 4.9277,C 0.1052,E1 4.8457,E2 329.5847} C_DIS
LIN {X -75.5458,Y 115.4658,Z 181,A 124.8066,B 4.9277,C 0.1081,E1 4.842,E2 328.0083} C_DIS
LIN {X -78.4429,Y 113.5177,Z 181,A 126.4199,B 4.9277,C 0.1089,E1 4.8382,E2 326.3758} C_DIS
LIN {X -82.0886,Y 110.9098,Z 181,A 128.1753,B 4.9275,C 0.1129,E1 4.8343,E2 324.635} C_DIS
LIN {X -84.9191,Y 108.7578,Z 181,A 129.768,B 4.9275,C 0.1144,E1 4.8307,E2 323.0291} C_DIS
LIN {X -88.3471,Y 105.9922,Z 181,A 131.6662,B 4.9275,C 0.1171,E1 4.8266,E2 321.1237} C_DIS
LIN {X -91.7612,Y 103.0505,Z 181,A 133.451,B 4.9273,C 0.1213,E1 4.8229,E2 319.3512} C_DIS
LIN {X -94.3966,Y 100.642,Z 181,A 134.9636,B 4.9273,C 0.1238,E1 4.8198,E2 317.836} C_DIS
LIN {X -96.9358,Y 98.1988,Z 181,A 136.5744,B 4.9273,C 0.1255,E1 4.8165,E2 316.2081} C_DIS
LIN {X -100.0622,Y 95.0112,Z 181,A 138.3775,B 4.9271,C 0.1296,E1 4.8131,E2 314.4128} C_DIS
LIN {X -102.4871,Y 92.3902,Z 181,A 139.8927,B 4.9271,C 0.1325,E1 4.8102,E2 312.8948} C_DIS
LIN {X -104.8729,Y 89.6728,Z 181,A 141.4148,B 4.927,C 0.1355,E1 4.8074,E2 311.3715} C_DIS
LIN {X -107.4953,Y 86.511,Z 181,A 143.2218,B 4.9269,C 0.1384,E1 4.8042,E2 309.5532} C_DIS
LIN {X -109.8724,Y 83.4723,Z 181,A 144.7992,B 4.9268,C 0.1422,E1 4.8015,E2 307.9802} C_DIS
LIN {X -111.9848,Y 80.6162,Z 181,A 146.4254,B 4.9268,C 0.1443,E1 4.7988,E2 306.3364} C_DIS
LIN {X -114.5774,Y 76.8863,Z 181,A 148.2102,B 4.9266,C 0.1495,E1 4.796,E2 304.5659} C_DIS
LIN {X -116.4488,Y 74.0219,Z 181,A 149.7106,B 4.9265,C 0.1523,E1 4.7938,E2 303.0567} C_DIS
LIN {X -118.3254,Y 70.9833,Z 181,A 151.3397,B 4.9264,C 0.1547,E1 4.7914,E2 301.4106} C_DIS
LIN {X -120.595,Y 67.0542,Z 181,A 153.1107,B 4.9262,C 0.1602,E1 4.7889,E2 299.6554} C_DIS
LIN {X -121.8009,Y 64.8378,Z 181,A 154.2245,B 4.9262,C 0.1623,E1 4.7875,E2 298.5342} C_DIS
LIN {X -123.5129,Y 61.5113,Z 181,A 155.6868,B 4.926,C 0.167,E1 4.7856,E2 297.0846} C_DIS
LIN {X -124.8765,Y 58.6978,Z 181,A 157.2681,B 4.926,C 0.1681,E1 4.7837,E2 295.469} C_DIS
LIN {X -126.5234,Y 55.0523,Z 181,A 158.8104,B 4.9258,C 0.1733,E1 4.782,E2 293.9429} C_DIS
LIN {X -127.6892,Y 52.2962,Z 181,A 160.1323,B 4.9257,C 0.176,E1 4.7805,E2 292.6122} C_DIS
LIN {X -128.9477,Y 49.1112,Z 181,A 161.5929,B 4.9256,C 0.1794,E1 4.7791,E2 291.148} C_DIS
LIN {X -130.1208,Y 45.913,Z 181,A 163.0459,B 4.9254,C 0.1829,E1 4.7777,E2 289.6913} C_DIS
LIN {X -131.1811,Y 42.7911,Z 181,A 164.5805,B 4.9254,C 0.1853,E1 4.7763,E2 288.137} C_DIS
LIN {X -132.2684,Y 39.2967,Z 181,A 165.9041,B 4.9251,C 0.191,E1 4.7753,E2 286.8393} C_DIS
LIN {X -133.1077,Y 36.3579,Z 181,A 167.351,B 4.9251,C 0.1931,E1 4.7742,E2 285.3711} C_DIS
LIN {X -133.9663,Y 33.0525,Z 181,A 168.743,B 4.9249,C 0.1972,E1 4.7732,E2 283.9835} C_DIS
LIN {X -134.7775,Y 29.5656,Z 181,A 170.1662,B 4.9247,C 0.2018,E1 4.7723,E2 282.5695} C_DIS
LIN {X -135.3904,Y 26.6247,Z 181,A 171.5872,B 4.9247,C 0.2039,E1 4.7715,E2 281.1276} C_DIS
LIN {X -135.9811,Y 23.4217,Z 181,A 172.9781,B 4.9245,C 0.2074,E1 4.7709,E2 279.7329} C_DIS
LIN {X -136.5386,Y 19.9066,Z 181,A 174.5038,B 4.9243,C 0.2112,E1 4.7702,E2 278.2024} C_DIS
LIN {X -136.9918,Y 16.4986,Z 181,A 175.9912,B 4.9241,C 0.2148,E1 4.7697,E2 276.7084} C_DIS
LIN {X -137.4258,Y 12.3985,Z 181,A 177.7268,B 4.9239,C 0.2194,E1 4.7692,E2 274.9712} C_DIS
LIN {X -137.6777,Y 9.1803,Z 181,A 179.1048,B 4.9238,C 0.2229,E1 4.7689,E2 273.5896} C_DIS
LIN {X -137.8675,Y 5.6182,Z 181,A -179.3181,B 4.9236,C 0.2264,E1 4.7687,E2 272.0013} C_DIS
LIN {X -137.9666,Y 2.0608,Z 181,A -177.7936,B 4.9235,C 0.2302,E1 4.7687,E2 270.4719} C_DIS
LIN {X -137.9741,Y -1.6104,Z 181,A -176.3121,B 4.9232,C 0.2349,E1 4.7687,E2 268.9971} C_DIS
LIN {X -137.9071,Y -4.6039,Z 181,A -174.997,B 4.9231,C 0.2379,E1 4.7687,E2 267.6738} C_DIS
LIN {X -137.7317,Y -8.3043,Z 181,A -173.3807,B 4.9229,C 0.2416,E1 4.769,E2 266.0486} C_DIS
LIN {X -137.5053,Y -11.4569,Z 181,A -172.204,B 4.9227,C 0.2464,E1 4.7692,E2 264.89} C_DIS
LIN {X -137.2746,Y -13.9732,Z 181,A -170.9406,B 4.9227,C 0.2477,E1 4.7696,E2 263.6002} C_DIS
LIN {X -136.9157,Y -17.1361,Z 181,A -169.6076,B 4.9224,C 0.2513,E1 4.77,E2 262.2666} C_DIS
LIN {X -136.428,Y -20.6523,Z 181,A -168.0319,B 4.9223,C 0.2546,E1 4.7707,E2 260.6788} C_DIS
LIN {X -135.8724,Y -24.0348,Z 181,A -166.6506,B 4.922,C 0.2589,E1 4.7713,E2 259.3039} C_DIS
LIN {X -135.3564,Y -26.797,Z 181,A -165.3691,B 4.922,C 0.2613,E1 4.772,E2 258.0085} C_DIS
LIN {X -134.6211,Y -30.2699,Z 181,A -163.8593,B 4.9217,C 0.2651,E1 4.7729,E2 256.4949} C_DIS
Enddeposition()
END
